// TIA Portal project "Synch Controller 20220313" (V15.1)

(* hardware
DEVICE "S71500/ET200MP station_1"  S7-1500 station
   slot 0: "导轨_0"  Rack  6ES7 590-1***0-0AA0
   slot 1: "PLC_1"  CPU 1516-3 PN/DP  6ES7 516-3AN01-0AB0  V2.6
      slot 3: "CPU 显示_1"  6ES7591-1BA00-0AA0
*)

// ===== PLC "PLC_1"  CPU 1516-3 PN/DP =====

VAR_GLOBAL   // PLC tag table "model"
   "left_cylinder_velocity" AT %MD200 : Real;
   "left_cylinder_position" AT %MD204 : Real;
   "right_cylinder_velocity" AT %MD208 : Real;
   "right_cylinder_position" AT %MD212 : Real;
   "left_cylinder_cmd[%]" AT %MD216 : Real;
   "right_cylinder_cmd[%]" AT %MD220 : Real;
   "model_run" AT %M100.0 : Bool;
   "left_cylinder_pos_init" AT %MD224 : Real;
   "right_cylinder_pos_init" AT %MD228 : Real;
END_VAR

VAR_GLOBAL   // PLC tag table "controller"
   "controller_run" AT %M300.1 : Bool;
   "ref_velocity" AT %MD400 : Real;
   "pos_loop_kp" AT %MD404 : Real;
   "pos_loop_Ti" AT %MD408 : Real;
   "vel_loop_kp" AT %MD412 : Real;
   "vel_loop_Ti" AT %MD416 : Real;
   "vel_loop_ff_kp" AT %MD420 : Real;
END_VAR

VAR_GLOBAL   // PLC tag table "test"
   "reset0" AT %M500.0 : Bool;
   "reset1" AT %M500.1 : Bool;
   "reset2" AT %M500.2 : Bool;
   "reset3" AT %M500.3 : Bool;
   "reset4" AT %M500.4 : Bool;
   "parameter1" AT %M500.6 : Bool;
   "parameter2" AT %M500.7 : Bool;
   "parameter3" AT %M501.0 : Bool;
   "parameter4" AT %M501.1 : Bool;
   "parameter5" AT %M501.2 : Bool;
   "autotest_run" AT %M500.5 : Bool;
   "seq_running" AT %M501.3 : Bool;
END_VAR

DATA_BLOCK "test_DB"   // DB3
{ S7_Optimized_Access := 'TRUE' }
VERSION : 0.1
// stored: InstanceOfName test
"test"
BEGIN
END_DATA_BLOCK

// folder: ctrl_synch/controller

DATA_BLOCK "controller_DB"   // DB9
{ S7_Optimized_Access := 'TRUE' }
VERSION : 0.1
// stored: InstanceOfName controller
"controller"
BEGIN
END_DATA_BLOCK

// folder: ctrl_synch/model

DATA_BLOCK "left_cylinder_DB"   // DB7
{ S7_Optimized_Access := 'TRUE' }
VERSION : 0.1
// stored: InstanceOfName cylinder
"cylinder"
BEGIN
END_DATA_BLOCK

DATA_BLOCK "right_cylinder_DB"   // DB8
{ S7_Optimized_Access := 'TRUE' }
VERSION : 0.1
// stored: InstanceOfName cylinder
"cylinder"
BEGIN
END_DATA_BLOCK

// folder: (top level)

FUNCTION_BLOCK "test"   // FB1, GRAPH_PLUS
{ S7_Optimized_Access := 'TRUE' }
VERSION : 0.1
   VAR_INPUT
      OFF_SQ : Bool := false;   // 关闭顺控器
      INIT_SQ : Bool := false;   // 将顺序设置为初始状态
      ACK_EF : Bool := false;   // 确认所有的错误和故障
      S_PREV : Bool := false;   // 在S_NO输出参数中显示前导步
      S_NEXT : Bool := false;   // 在S_NO输出参数中显示后续步。
      SW_AUTO : Bool := false;   // 自动模式
      SW_TAP : Bool := false;   // 半自动/转换条件切换
      SW_TOP : Bool := false;   // 半自动/忽略转换条件
      SW_MAN : Bool := false;   // 手动模式
      S_SEL : Int := 0;   // 选择要在 S_NO中输出的步。
      S_ON : Bool := false;   // 激活S_NO 中显示的步。
      S_OFF : Bool := false;   // 取消激活 S_NO 中标识的步
      T_PUSH : Bool := false;   // 允许在半自动模式下跳过转换条件。
   END_VAR
   VAR_OUTPUT
      S_NO : Int := 0;   // 步编号
      S_MORE : Bool := false;   // 更多步可用，并可在S_NO中显示。
      S_ACTIVE : Bool := false;   // 在S_NO 中显示的步是激活的。
      ERR_FLT : Bool := false;   // 互锁条件或监控条件组出错
      AUTO_ON : Bool := false;   // 当前为自动模式
      TAP_ON : Bool := false;   // 已启用SW_TAP模式。
      TOP_ON : Bool := false;   // 启用半自动模式/忽略转换条件。
      MAN_ON : Bool := false;   // 已启用手动模式。
      reset0 : Bool;   // initial status
      parameter1 : Bool;
      reset1 : Bool;
      parameter2 : Bool;
      reset2 : Bool;
      parameter3 : Bool;
      reset3 : Bool;
      parameter4 : Bool;
      reset4 : Bool;
      parameter5 : Bool;
   END_VAR
   VAR
      HMI_INFO : Array[0..8] of UInt;
      IF_PAR : G7_IfParPlus_V6;
      RT_DATA : G7_RTDataPlus_V6;   // 内部数据区
      Trans1 : G7_TransitionPlus_V6;   // 转换结构
      Trans2 : G7_TransitionPlus_V6;   // 转换结构
      Trans3 : G7_TransitionPlus_V6;   // 转换结构
      Trans4 : G7_TransitionPlus_V6;   // 转换结构
      Trans5 : G7_TransitionPlus_V6;   // 转换结构
      Trans6 : G7_TransitionPlus_V6;   // 转换结构
      Trans7 : G7_TransitionPlus_V6;   // 转换结构
      Trans8 : G7_TransitionPlus_V6;   // 转换结构
      Trans9 : G7_TransitionPlus_V6;   // 转换结构
      Trans10 : G7_TransitionPlus_V6;   // 转换结构
      Step1 : G7_StepPlus_V6;   // 步结构
      Step2 : G7_StepPlus_V6;   // 步结构
      Step3 : G7_StepPlus_V6;   // 步结构
      Step4 : G7_StepPlus_V6;   // 步结构
      Step5 : G7_StepPlus_V6;   // 步结构
      Step6 : G7_StepPlus_V6;   // 步结构
      Step7 : G7_StepPlus_V6;   // 步结构
      Step8 : G7_StepPlus_V6;   // 步结构
      Step9 : G7_StepPlus_V6;   // 步结构
      Step10 : G7_StepPlus_V6;   // 步结构
      SINI : Array[0..1] of USInt;
      LSTT : Array[0..9] of USInt;
      ATAJ : Array[0..9] of USInt;
      ATAB : Array[0..9] of USInt;
      PSTT : Array[0..9] of USInt;
      NSTT : Array[0..9] of USInt;
      ASSJ : Array[0..9] of USInt;
      ASSB : Array[0..9] of USInt;
      PTTS : Array[0..9] of USInt;
      NTTS : Array[0..9] of USInt;
      SW_SQTS : Array[0..9] of USInt;
      SWITCH : Array[0..0] of USInt;
      TVX : Array[0..1] of USInt;
      TTX : Array[0..1] of USInt;
      TSX : Array[0..1] of USInt;
      S00X : Array[0..1] of USInt;
      SOFFX : Array[0..1] of USInt;
      SONX : Array[0..1] of USInt;
      SAX : Array[0..1] of USInt;
      SERRX : Array[0..10] of USInt;
      SMX : Array[0..10] of USInt;
      S0X : Array[0..10] of USInt;
      S1X : Array[0..10] of USInt;
      IL_ALARM_INST : Diag_Alarm;
      SUP_ALARM_INST : Diag_Alarm;
      STEP_TIME_ALARM_INST : Diag_Alarm;
      IEC_TIMER_INST : IEC_TIMER;
      TRANSACTION_FLAG : Bool := false;
   END_VAR
   VAR CONSTANT
      MIN_INTERVAL : Time := T#10ms;
      MAX_INTERVAL : Time := T#40s;
      LAST_INTERVAL : Time := T#60s;
   END_VAR
   // SINI[0] := 2;
   // LSTT[0] := 255;
   // LSTT[1] := 255;
   // LSTT[2] := 255;
   // LSTT[3] := 255;
   // LSTT[4] := 255;
   // LSTT[5] := 255;
   // LSTT[6] := 255;
   // LSTT[7] := 255;
   // ATAJ[1] := 1;
   // ATAJ[2] := 2;
   // ATAJ[3] := 3;
   // ATAJ[4] := 4;
   // ATAJ[5] := 5;
   // ATAJ[6] := 6;
   // ATAJ[7] := 7;
   // ATAJ[8] := 8;
   // ATAB[1] := 1;
   // ATAB[2] := 2;
   // ATAB[3] := 3;
   // ATAB[4] := 4;
   // ATAB[5] := 5;
   // ATAB[6] := 6;
   // ATAB[7] := 7;
   // ATAB[8] := 8;
   // PSTT[1] := 1;
   // PSTT[2] := 2;
   // PSTT[3] := 3;
   // PSTT[4] := 4;
   // PSTT[5] := 5;
   // PSTT[6] := 6;
   // PSTT[7] := 7;
   // PSTT[8] := 8;
   // NSTT[0] := 1;
   // NSTT[1] := 2;
   // NSTT[2] := 3;
   // NSTT[3] := 4;
   // NSTT[4] := 5;
   // NSTT[5] := 6;
   // NSTT[6] := 7;
   // NSTT[7] := 8;
   // ASSJ[1] := 1;
   // ASSJ[2] := 2;
   // ASSJ[3] := 3;
   // ASSJ[4] := 4;
   // ASSJ[5] := 5;
   // ASSJ[6] := 6;
   // ASSJ[7] := 7;
   // ASSJ[8] := 8;
   // ASSB[1] := 1;
   // ASSB[2] := 2;
   // ASSB[3] := 3;
   // ASSB[4] := 4;
   // ASSB[5] := 5;
   // ASSB[6] := 6;
   // ASSB[7] := 7;
   // ASSB[8] := 8;
   // PTTS[0] := 255;
   // PTTS[2] := 1;
   // PTTS[3] := 2;
   // PTTS[4] := 3;
   // PTTS[5] := 4;
   // PTTS[6] := 5;
   // PTTS[7] := 6;
   // PTTS[8] := 7;
   // NTTS[1] := 1;
   // NTTS[2] := 2;
   // NTTS[3] := 3;
   // NTTS[4] := 4;
   // NTTS[5] := 5;
   // NTTS[6] := 6;
   // NTTS[7] := 7;
   // NTTS[8] := 8;
   // TVX[0] := 16#1;
   // TTX[0] := 16#1;
   // TSX[0] := 16#1;
   // S00X[0] := 16#1;
   // SOFFX[0] := 16#1;
   // SONX[0] := 16#1;
   // SAX[0] := 16#1;
   // SERRX[0] := 16#1;
   // SMX[0] := 16#1;
   // S0X[0] := 16#1;
   // S1X[0] := 16#1;
   // LSTT[8] := 255;
   // ATAJ[9] := 9;
   // ATAB[9] := 9;
   // PSTT[9] := 9;
   // NSTT[8] := 9;
   // ASSJ[9] := 9;
   // ASSB[9] := 9;
   // PTTS[9] := 8;
   // NTTS[9] := 9;
BEGIN
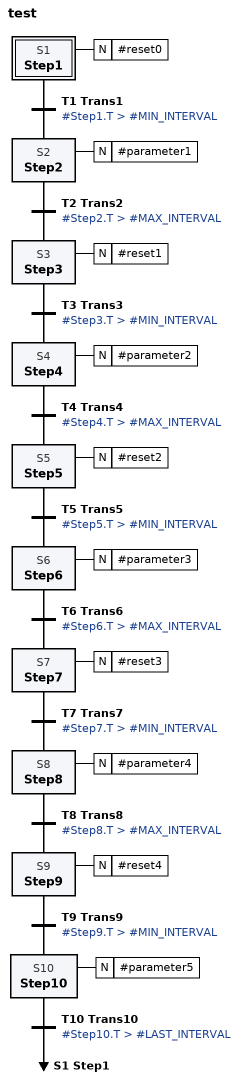
   // sequencer 1
   INITIAL_STEP Step1:   // S1, max time T#10S, warning time T#7S
              N    #reset0
   END_STEP
   TRANSITION Trans1 FROM Step1 TO Step2   // T1
      := #Step1.T > #MIN_INTERVAL;
   END_TRANSITION
   STEP Step2:   // S2, max time T#10S, warning time T#7S
              N    #parameter1
   END_STEP
   TRANSITION Trans2 FROM Step2 TO Step3   // T2
      := #Step2.T > #MAX_INTERVAL;
   END_TRANSITION
   STEP Step3:   // S3, max time T#10S, warning time T#7S
              N    #reset1
   END_STEP
   TRANSITION Trans3 FROM Step3 TO Step4   // T3
      := #Step3.T > #MIN_INTERVAL;
   END_TRANSITION
   STEP Step4:   // S4, max time T#10S, warning time T#7S
              N    #parameter2
   END_STEP
   TRANSITION Trans4 FROM Step4 TO Step5   // T4
      := #Step4.T > #MAX_INTERVAL;
   END_TRANSITION
   STEP Step5:   // S5, max time T#10S, warning time T#7S
              N    #reset2
   END_STEP
   TRANSITION Trans5 FROM Step5 TO Step6   // T5
      := #Step5.T > #MIN_INTERVAL;
   END_TRANSITION
   STEP Step6:   // S6, max time T#10S, warning time T#7S
              N    #parameter3
   END_STEP
   TRANSITION Trans6 FROM Step6 TO Step7   // T6
      := #Step6.T > #MAX_INTERVAL;
   END_TRANSITION
   STEP Step7:   // S7, max time T#10S, warning time T#7S
              N    #reset3
   END_STEP
   TRANSITION Trans7 FROM Step7 TO Step8   // T7
      := #Step7.T > #MIN_INTERVAL;
   END_TRANSITION
   STEP Step8:   // S8, max time T#10S, warning time T#7S
              N    #parameter4
   END_STEP
   TRANSITION Trans8 FROM Step8 TO Step9   // T8
      := #Step8.T > #MAX_INTERVAL;
   END_TRANSITION
   STEP Step9:   // S9, max time T#10S, warning time T#7S
              N    #reset4
   END_STEP
   TRANSITION Trans9 FROM Step9 TO Step10   // T9
      := #Step9.T > #MIN_INTERVAL;
   END_TRANSITION
   STEP Step10:   // S10, max time T#10S, warning time T#7S
              N    #parameter5
   END_STEP
   TRANSITION Trans10 FROM Step10 TO Step1   // T10, jump
      := #Step10.T > #LAST_INTERVAL;
   END_TRANSITION
END_FUNCTION_BLOCK

ORGANIZATION_BLOCK "Main"   // OB1, LAD, ProgramCycle
TITLE = "Main Program Sweep (Cycle)"
{ S7_Optimized_Access := 'TRUE' }
VERSION : 0.1
   VAR_INPUT
      Initial_Call : Bool;   // Initial call of this OB
      Remanence : Bool;   // =True, if remanent data are available
   END_VAR
BEGIN

REGION Network 1
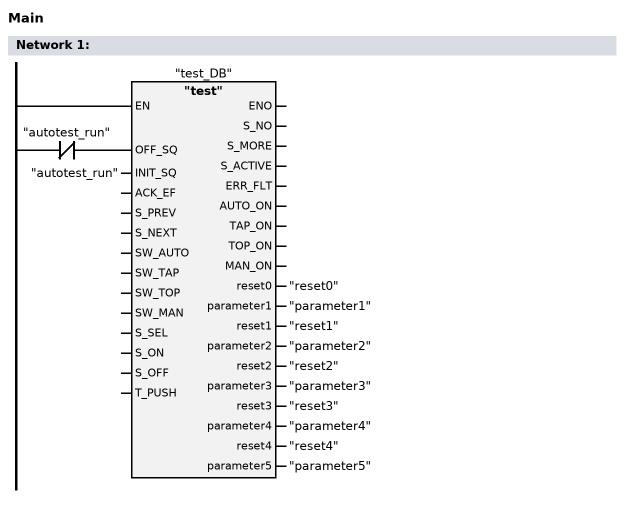
   RUNG wire#powerrail
      "test_DB"(OFF_SQ := wire#w1, INIT_SQ := "autotest_run", ACK_EF :=, S_PREV :=, S_NEXT :=, SW_AUTO :=, SW_TAP :=, SW_TOP :=, SW_MAN :=, S_SEL :=, S_ON :=, S_OFF :=, T_PUSH :=, S_NO =>, S_MORE =>, S_ACTIVE =>, ERR_FLT =>, AUTO_ON =>, TAP_ON =>, TOP_ON =>, MAN_ON =>, reset0 => "reset0", parameter1 => "parameter1", reset1 => "reset1", parameter2 => "parameter2", reset2 => "reset2", parameter3 => "parameter3", reset3 => "reset3", parameter4 => "parameter4", reset4 => "reset4", parameter5 => "parameter5")
   END_RUNG
   RUNG wire#powerrail
      I_Contact( "autotest_run" )
   END_RUNG wire#w1
   // the same network as SCL:
   "test_DB"(OFF_SQ := NOT "autotest_run",   // "test"
             INIT_SQ := "autotest_run",
             reset0 => "reset0",
             parameter1 => "parameter1",
             reset1 => "reset1",
             parameter2 => "parameter2",
             reset2 => "reset2",
             parameter3 => "parameter3",
             reset3 => "reset3",
             parameter4 => "parameter4",
             reset4 => "reset4",
             parameter5 => "parameter5");
END_REGION

REGION Network 2 (SCL): test-1
   // rated speed of cylinder = 50mm/s [100% openning of valve]
   // only position loop
   // IF ("reset0" OR
   //     "reset1" OR
   //     "reset2" OR
   //     "reset3" OR
   //     "reset4")OR
   //     NOT "autotest_run"
   // THEN
   //     "left_cylinder_pos_init" :=1100.0;
   //     "right_cylinder_pos_init" :=900.0;
   //     "ref_velocity" := 0.0;
   //     "model_run" := FALSE;
   //     "controller_run" := FALSE;
   // END_IF;

   // IF "parameter1" THEN
   //     "model_run" := TRUE;
   //     "controller_run" := TRUE;

   //     "ref_velocity" := 0.0;
   //     "pos_loop_kp" := 1.0;
   //     "pos_loop_Ti" := 0.0;
   //     "vel_loop_kp" := 0.0;
   //     "vel_loop_Ti" := 0.0;
   //     "vel_loop_ff_kp" := 1.0;

   // END_IF;


   // IF "parameter2" THEN
   //     "model_run" := TRUE;
   //     "controller_run" := TRUE;

   //     "ref_velocity" := 0.0;
   //     "pos_loop_kp" := 5.0;
   //     "pos_loop_Ti" := 0.0;
   //     "vel_loop_kp" := 0.0;
   //     "vel_loop_Ti" := 0.0;
   //     "vel_loop_ff_kp" := 1.0;

   // END_IF;

   // IF "parameter3" THEN
   //     "model_run" := TRUE;
   //     "controller_run" := TRUE;

   //     "ref_velocity" := 0.0;
   //     "pos_loop_kp" := 10.0;
   //     "pos_loop_Ti" := 0.0;
   //     "vel_loop_kp" := 0.0;
   //     "vel_loop_Ti" := 0.0;
   //     "vel_loop_ff_kp" := 1.0;

   // END_IF;

   // IF "parameter4" THEN
   //     "model_run" := TRUE;
   //     "controller_run" := TRUE;

   //     "ref_velocity" := 0.0;
   //     "pos_loop_kp" := 15.0;
   //     "pos_loop_Ti" := 0.0;
   //     "vel_loop_kp" := 0.0;
   //     "vel_loop_Ti" := 0.0;
   //     "vel_loop_ff_kp" := 1.0;

   // END_IF;

   // IF "parameter5" THEN
   //     "model_run" := TRUE;
   //     "controller_run" := TRUE;

   //     "ref_velocity" := 0.0;
   //     "pos_loop_kp" := 20.0;
   //     "pos_loop_Ti" := 0.0;
   //     "vel_loop_kp" := 0.0;
   //     "vel_loop_Ti" := 0.0;
   //     "vel_loop_ff_kp" := 1.0;

   // END_IF;
END_REGION

REGION Network 3 (SCL): test-2
   // rated speed of cylinder = 50mm/s [100% openning of valve]
   // position loop+velocity loop
   // IF ("reset0" OR
   //     "reset1" OR
   //     "reset2" OR
   //     "reset3" OR
   //     "reset4")OR
   //     NOT "autotest_run"
   // THEN
   //     "left_cylinder_pos_init" :=1100.0;
   //     "right_cylinder_pos_init" :=900.0;
   //     "ref_velocity" := 0.0;
   //     "model_run" := FALSE;
   //     "controller_run" := FALSE;
   // END_IF;
   // // 
   // IF "parameter1" THEN
   //     "model_run" := TRUE;
   //     "controller_run" := TRUE;

   //     "ref_velocity" := 0.0;
   //     "pos_loop_kp" := 1.0;
   //     "pos_loop_Ti" := 0.0;
   //     "vel_loop_kp" := 1.0;
   //     "vel_loop_Ti" := 0.0;
   //     "vel_loop_ff_kp" := 0.0;

   // END_IF;

   // // 
   // IF "parameter2" THEN
   //     "model_run" := TRUE;
   //     "controller_run" := TRUE;

   //     "ref_velocity" := 0.0;
   //     "pos_loop_kp" := 5.0;
   //     "pos_loop_Ti" := 0.0;
   //     "vel_loop_kp" := 1.0;
   //     "vel_loop_Ti" := 0.0;
   //     "vel_loop_ff_kp" := 0.0;

   // END_IF;
   // // 
   // IF "parameter3" THEN
   //     "model_run" := TRUE;
   //     "controller_run" := TRUE;

   //     "ref_velocity" := 0.0;
   //     "pos_loop_kp" := 10.0;
   //     "pos_loop_Ti" := 0.0;
   //     "vel_loop_kp" := 1.0;
   //     "vel_loop_Ti" := 0.0;
   //     "vel_loop_ff_kp" := 0.0;

   // END_IF;
   // //
   // IF "parameter4" THEN
   //     "model_run" := TRUE;
   //     "controller_run" := TRUE;

   //     "ref_velocity" := 0.0;
   //     "pos_loop_kp" := 15.0;
   //     "pos_loop_Ti" := 0.0;
   //     "vel_loop_kp" := 1.0;
   //     "vel_loop_Ti" := 0.0;
   //     "vel_loop_ff_kp" := 0.0;

   // END_IF;
   // //
   // IF "parameter5" THEN
   //     "model_run" := TRUE;
   //     "controller_run" := TRUE;

   //     "ref_velocity" := 0.0;
   //     "pos_loop_kp" := 20.0;
   //     "pos_loop_Ti" := 0.0;
   //     "vel_loop_kp" := 1.0;
   //     "vel_loop_Ti" := 0.0;
   //     "vel_loop_ff_kp" := 0.0;

   // END_IF;
END_REGION

REGION Network 4 (SCL): test-3
   // rated speed of cylinder = 50mm/s [100% openning of valve]
   // position loop+velocity loop+FF
   // IF ("reset0" OR
   //     "reset1" OR
   //     "reset2" OR
   //     "reset3" OR
   //     "reset4")OR
   //     NOT "autotest_run"
   // THEN
   //     "left_cylinder_pos_init" :=1100.0;
   //     "right_cylinder_pos_init" :=900.0;
   //     "ref_velocity" := 0.0;
   //     "model_run" := FALSE;
   //     "controller_run" := FALSE;
   // END_IF;
   // // 
   // IF "parameter1" THEN
   //     "model_run" := TRUE;
   //     "controller_run" := TRUE;

   //     "ref_velocity" := 0.0;
   //     "pos_loop_kp" := 1.0;
   //     "pos_loop_Ti" := 0.0;
   //     "vel_loop_kp" := 1.0;
   //     "vel_loop_Ti" := 0.0;
   //     "vel_loop_ff_kp" := 1.0;

   // END_IF;

   // // 
   // IF "parameter2" THEN
   //     "model_run" := TRUE;
   //     "controller_run" := TRUE;

   //     "ref_velocity" := 0.0;
   //     "pos_loop_kp" := 5.0;
   //     "pos_loop_Ti" := 0.0;
   //     "vel_loop_kp" := 1.0;
   //     "vel_loop_Ti" := 0.0;
   //     "vel_loop_ff_kp" := 1.0;

   // END_IF;
   // // 
   // IF "parameter3" THEN
   //     "model_run" := TRUE;
   //     "controller_run" := TRUE;

   //     "ref_velocity" := 0.0;
   //     "pos_loop_kp" := 10.0;
   //     "pos_loop_Ti" := 0.0;
   //     "vel_loop_kp" := 1.0;
   //     "vel_loop_Ti" := 0.0;
   //     "vel_loop_ff_kp" := 1.0;

   // END_IF;
   // //
   // IF "parameter4" THEN
   //     "model_run" := TRUE;
   //     "controller_run" := TRUE;

   //     "ref_velocity" := 0.0;
   //     "pos_loop_kp" := 15.0;
   //     "pos_loop_Ti" := 0.0;
   //     "vel_loop_kp" := 1.0;
   //     "vel_loop_Ti" := 0.0;
   //     "vel_loop_ff_kp" := 1.0;

   // END_IF;
   // //
   // IF "parameter5" THEN
   //     "model_run" := TRUE;
   //     "controller_run" := TRUE;

   //     "ref_velocity" := 0.0;
   //     "pos_loop_kp" := 20.0;
   //     "pos_loop_Ti" := 0.0;
   //     "vel_loop_kp" := 1.0;
   //     "vel_loop_Ti" := 0.0;
   //     "vel_loop_ff_kp" := 1.0;

   // END_IF;
END_REGION

REGION Network 5 (SCL): test-4
   // velocity loop
   // IF ("reset0" OR
   //     "reset1" OR
   //     "reset2" OR
   //     "reset3" OR
   //     "reset4")OR
   //     NOT "autotest_run"
   // THEN
   //     "left_cylinder_pos_init" :=1000.0;
   //     "right_cylinder_pos_init" :=1000.0;
   //     "ref_velocity" := 0.0;
   //     "model_run" := FALSE;
   //     "controller_run" := FALSE;
   // END_IF;
   // // 
   // IF "parameter1" THEN
   //     "model_run" := TRUE;
   //     "controller_run" := TRUE;

   //     "ref_velocity" := 40.0;
   //     "pos_loop_kp" := 10.0;
   //     "pos_loop_Ti" := 0.0;
   //     "vel_loop_kp" := 1.0;
   //     "vel_loop_Ti" := 0.0;
   //     "vel_loop_ff_kp" := 0.0;

   // END_IF;

   // // 
   // IF "parameter2" THEN
   //     "model_run" := TRUE;
   //     "controller_run" := TRUE;

   //     "ref_velocity" := 40.0;
   //     "pos_loop_kp" := 10.0;
   //     "pos_loop_Ti" := 0.0;
   //     "vel_loop_kp" := 2.0;
   //     "vel_loop_Ti" := 0.0;
   //     "vel_loop_ff_kp" := 1.0;

   // END_IF;
   // // 
   // IF "parameter3" THEN
   //     "model_run" := TRUE;
   //     "controller_run" := TRUE;

   //     "ref_velocity" := 40.0;
   //     "pos_loop_kp" := 10.0;
   //     "pos_loop_Ti" := 0.0;
   //     "vel_loop_kp" := 5.0;
   //     "vel_loop_Ti" := 0.0;
   //     "vel_loop_ff_kp" := 0.0;

   // END_IF;
   // //
   // IF "parameter4" THEN
   //     "model_run" := TRUE;
   //     "controller_run" := TRUE;

   //     "ref_velocity" := 40.0;
   //     "pos_loop_kp" := 10.0;
   //     "pos_loop_Ti" := 0.0;
   //     "vel_loop_kp" := 10.0;
   //     "vel_loop_Ti" := 0.0;
   //     "vel_loop_ff_kp" := 0.0;

   // END_IF;
   // //
   // IF "parameter5" THEN
   //     "model_run" := TRUE;
   //     "controller_run" := TRUE;

   //     "ref_velocity" := 40.0;
   //     "pos_loop_kp" := 10.0;
   //     "pos_loop_Ti" := 0.0;
   //     "vel_loop_kp" := 20.0;
   //     "vel_loop_Ti" := 0.0;
   //     "vel_loop_ff_kp" := 0.0;

   // END_IF;
END_REGION

REGION Network 6 (SCL): test-5
   // velocity loop
   // IF ("reset0" OR
   //     "reset1" OR
   //     "reset2" OR
   //     "reset3" OR
   //     "reset4")OR
   //     NOT "autotest_run"
   // THEN
   //     "left_cylinder_pos_init" :=1000.0;
   //     "right_cylinder_pos_init" :=1000.0;
   //     "ref_velocity" := 0.0;
   //     "model_run" := FALSE;
   //     "controller_run" := FALSE;
   // END_IF;
   // // 
   // IF "parameter1" THEN
   //     "model_run" := TRUE;
   //     "controller_run" := TRUE;

   //     "ref_velocity" := 40.0;
   //     "pos_loop_kp" := 10.0;
   //     "pos_loop_Ti" := 0.0;
   //     "vel_loop_kp" := 1.0;
   //     "vel_loop_Ti" := 1.0;
   //     "vel_loop_ff_kp" := 0.0;

   // END_IF;

   // // 
   // IF "parameter2" THEN
   //     "model_run" := TRUE;
   //     "controller_run" := TRUE;

   //     "ref_velocity" := 40.0;
   //     "pos_loop_kp" := 10.0;
   //     "pos_loop_Ti" := 0.0;
   //     "vel_loop_kp" := 2.0;
   //     "vel_loop_Ti" := 1.0;
   //     "vel_loop_ff_kp" := 1.0;

   // END_IF;
   // // 
   // IF "parameter3" THEN
   //     "model_run" := TRUE;
   //     "controller_run" := TRUE;

   //     "ref_velocity" := 40.0;
   //     "pos_loop_kp" := 10.0;
   //     "pos_loop_Ti" := 0.0;
   //     "vel_loop_kp" := 5.0;
   //     "vel_loop_Ti" := 1.0;
   //     "vel_loop_ff_kp" := 0.0;

   // END_IF;
   // //
   // IF "parameter4" THEN
   //     "model_run" := TRUE;
   //     "controller_run" := TRUE;

   //     "ref_velocity" := 40.0;
   //     "pos_loop_kp" := 10.0;
   //     "pos_loop_Ti" := 0.0;
   //     "vel_loop_kp" := 10.0;
   //     "vel_loop_Ti" := 1.0;
   //     "vel_loop_ff_kp" := 0.0;

   // END_IF;
   // //
   // IF "parameter5" THEN
   //     "model_run" := TRUE;
   //     "controller_run" := TRUE;

   //     "ref_velocity" := 40.0;
   //     "pos_loop_kp" := 10.0;
   //     "pos_loop_Ti" := 0.0;
   //     "vel_loop_kp" := 20.0;
   //     "vel_loop_Ti" := 1.0;
   //     "vel_loop_ff_kp" := 0.0;

   // END_IF;
END_REGION

REGION Network 7 (SCL): test-5
   // velocity loop
   // IF ("reset0" OR
   //     "reset1" OR
   //     "reset2" OR
   //     "reset3" OR
   //     "reset4")OR
   //     NOT "autotest_run"
   // THEN
   //     "left_cylinder_pos_init" :=1000.0;
   //     "right_cylinder_pos_init" :=1000.0;
   //     "ref_velocity" := 0.0;
   //     "model_run" := FALSE;
   //     "controller_run" := FALSE;
   // END_IF;

   // IF "parameter1" THEN
   //     "model_run" := TRUE;
   //     "controller_run" := TRUE;

   //     "ref_velocity" := 40.0;
   //     "pos_loop_kp" := 10.0;
   //     "pos_loop_Ti" := 0.0;
   //     "vel_loop_kp" := 1.0;
   //     "vel_loop_Ti" := 10.0;
   //     "vel_loop_ff_kp" := 0.0;

   // END_IF;


   // IF "parameter2" THEN
   //     "model_run" := TRUE;
   //     "controller_run" := TRUE;

   //     "ref_velocity" := 40.0;
   //     "pos_loop_kp" := 10.0;
   //     "pos_loop_Ti" := 0.0;
   //     "vel_loop_kp" := 2.0;
   //     "vel_loop_Ti" := 10.0;
   //     "vel_loop_ff_kp" := 0.0;

   // END_IF;

   // IF "parameter3" THEN
   //     "model_run" := TRUE;
   //     "controller_run" := TRUE;

   //     "ref_velocity" := 40.0;
   //     "pos_loop_kp" := 10.0;
   //     "pos_loop_Ti" := 0.0;
   //     "vel_loop_kp" := 5.0;
   //     "vel_loop_Ti" := 10.0;
   //     "vel_loop_ff_kp" := 0.0;

   // END_IF;

   // IF "parameter4" THEN
   //     "model_run" := TRUE;
   //     "controller_run" := TRUE;

   //     "ref_velocity" := 40.0;
   //     "pos_loop_kp" := 10.0;
   //     "pos_loop_Ti" := 0.0;
   //     "vel_loop_kp" := 10.0;
   //     "vel_loop_Ti" := 10.0;
   //     "vel_loop_ff_kp" := 0.0;

   // END_IF;

   // IF "parameter5" THEN
   //     "model_run" := TRUE;
   //     "controller_run" := TRUE;

   //     "ref_velocity" := 40.0;
   //     "pos_loop_kp" := 10.0;
   //     "pos_loop_Ti" := 0.0;
   //     "vel_loop_kp" := 20.0;
   //     "vel_loop_Ti" := 10.0;
   //     "vel_loop_ff_kp" := 0.0;

   // END_IF;
END_REGION

REGION Network 8 (SCL): test-7
   // velocity loop
   // IF ("reset0" OR
   //     "reset1" OR
   //     "reset2" OR
   //     "reset3" OR
   //     "reset4")OR
   //     NOT "autotest_run"
   // THEN
   //     "left_cylinder_pos_init" :=1000.0;
   //     "right_cylinder_pos_init" :=1000.0;
   //     "ref_velocity" := 0.0;
   //     "model_run" := FALSE;
   //     "controller_run" := FALSE;
   // END_IF;
   // // 
   // IF "parameter1" THEN
   //     "model_run" := TRUE;
   //     "controller_run" := TRUE;

   //     "ref_velocity" := 40.0;
   //     "pos_loop_kp" := 10.0;
   //     "pos_loop_Ti" := 0.0;
   //     "vel_loop_kp" := 1.0;
   //     "vel_loop_Ti" := 1.0;
   //     "vel_loop_ff_kp" := 0.0;

   // END_IF;

   // // 
   // IF "parameter2" THEN
   //     "model_run" := TRUE;
   //     "controller_run" := TRUE;

   //     "ref_velocity" := 40.0;
   //     "pos_loop_kp" := 10.0;
   //     "pos_loop_Ti" := 0.0;
   //     "vel_loop_kp" := 2.0;
   //     "vel_loop_Ti" := 1.0;
   //     "vel_loop_ff_kp" := 0.0;

   // END_IF;
   // // 
   // IF "parameter3" THEN
   //     "model_run" := TRUE;
   //     "controller_run" := TRUE;

   //     "ref_velocity" := 40.0;
   //     "pos_loop_kp" := 10.0;
   //     "pos_loop_Ti" := 0.0;
   //     "vel_loop_kp" := 2.0;
   //     "vel_loop_Ti" := 2.0;
   //     "vel_loop_ff_kp" := 0.0;

   // END_IF;
   // //
   // IF "parameter4" THEN
   //     "model_run" := TRUE;
   //     "controller_run" := TRUE;

   //     "ref_velocity" := 40.0;
   //     "pos_loop_kp" := 10.0;
   //     "pos_loop_Ti" := 0.0;
   //     "vel_loop_kp" := 5.0;
   //     "vel_loop_Ti" := 5.0;
   //     "vel_loop_ff_kp" := 0.0;

   // END_IF;
   // //
   // IF "parameter5" THEN
   //     "model_run" := TRUE;
   //     "controller_run" := TRUE;

   //     "ref_velocity" := 40.0;
   //     "pos_loop_kp" := 10.0;
   //     "pos_loop_Ti" := 0.0;
   //     "vel_loop_kp" := 5.0;
   //     "vel_loop_Ti" := 10.0;
   //     "vel_loop_ff_kp" := 0.0;

   // END_IF;
END_REGION

REGION Network 9 (SCL): test-9
   // velocity loop
   // IF ("reset0" OR
   //     "reset1" OR
   //     "reset2" OR
   //     "reset3" OR
   //     "reset4")OR
   //     NOT "autotest_run"
   // THEN
   //     "left_cylinder_pos_init" :=1100.0;
   //     "right_cylinder_pos_init" :=900.0;
   //     "ref_velocity" := 0.0;
   //     "model_run" := FALSE;
   //     "controller_run" := FALSE;
   // END_IF;
   // // 
   // IF "parameter1" THEN
   //     "model_run" := TRUE;
   //     "controller_run" := TRUE;

   //     "ref_velocity" := 0.0;
   //     "pos_loop_kp" := 10.0;
   //     "pos_loop_Ti" := 0.0;
   //     "vel_loop_kp" := 1.0;
   //     "vel_loop_Ti" := 1.0;
   //     "vel_loop_ff_kp" := 0.0;

   // END_IF;

   // // 
   // IF "parameter2" THEN
   //     "model_run" := TRUE;
   //     "controller_run" := TRUE;

   //     "ref_velocity" := 0.0;
   //     "pos_loop_kp" := 10.0;
   //     "pos_loop_Ti" := 0.0;
   //     "vel_loop_kp" := 2.0;
   //     "vel_loop_Ti" := 1.0;
   //     "vel_loop_ff_kp" := 0.0;

   // END_IF;
   // // 
   // IF "parameter3" THEN
   //     "model_run" := TRUE;
   //     "controller_run" := TRUE;

   //     "ref_velocity" := 0.0;
   //     "pos_loop_kp" := 10.0;
   //     "pos_loop_Ti" := 0.0;
   //     "vel_loop_kp" := 2.0;
   //     "vel_loop_Ti" := 2.0;
   //     "vel_loop_ff_kp" := 0.0;

   // END_IF;
   // //
   // IF "parameter4" THEN
   //     "model_run" := TRUE;
   //     "controller_run" := TRUE;

   //     "ref_velocity" := 0.0;
   //     "pos_loop_kp" := 10.0;
   //     "pos_loop_Ti" := 0.0;
   //     "vel_loop_kp" := 5.0;
   //     "vel_loop_Ti" := 5.0;
   //     "vel_loop_ff_kp" := 0.0;

   // END_IF;
   // //
   // IF "parameter5" THEN
   //     "model_run" := TRUE;
   //     "controller_run" := TRUE;

   //     "ref_velocity" := 0.0;
   //     "pos_loop_kp" := 10.0;
   //     "pos_loop_Ti" := 0.0;
   //     "vel_loop_kp" := 5.0;
   //     "vel_loop_Ti" := 10.0;
   //     "vel_loop_ff_kp" := 0.0;

   // END_IF;
END_REGION

REGION Network 10 (SCL): test-10
   // velocity loop
   // IF ("reset0" OR
   //     "reset1" OR
   //     "reset2" OR
   //     "reset3" OR
   //     "reset4")OR
   //     NOT "autotest_run"
   // THEN
   //     "left_cylinder_pos_init" :=1100.0;
   //     "right_cylinder_pos_init" :=900.0;
   //     "ref_velocity" := 0.0;
   //     "model_run" := FALSE;
   //     "controller_run" := FALSE;
   // END_IF;
   // // 
   // IF "parameter1" THEN
   //     "model_run" := TRUE;
   //     "controller_run" := TRUE;

   //     "ref_velocity" := 0.0;
   //     "pos_loop_kp" := 5.0;
   //     "pos_loop_Ti" := 0.0;
   //     "vel_loop_kp" := 2.0;
   //     "vel_loop_Ti" := 5.0;
   //     "vel_loop_ff_kp" := 0.0;

   // END_IF;

   // // 
   // IF "parameter2" THEN
   //     "model_run" := TRUE;
   //     "controller_run" := TRUE;

   //     "ref_velocity" := 0.0;
   //     "pos_loop_kp" := 5.0;
   //     "pos_loop_Ti" := 0.0;
   //     "vel_loop_kp" := 2.0;
   //     "vel_loop_Ti" := 10.0;
   //     "vel_loop_ff_kp" := 0.0;

   // END_IF;
   // // 
   // IF "parameter3" THEN
   //     "model_run" := TRUE;
   //     "controller_run" := TRUE;

   //     "ref_velocity" := 0.0;
   //     "pos_loop_kp" := 2.0;
   //     "pos_loop_Ti" := 0.0;
   //     "vel_loop_kp" := 2.0;
   //     "vel_loop_Ti" := 5.0;
   //     "vel_loop_ff_kp" := 0.0;

   // END_IF;
   // //
   // IF "parameter4" THEN
   //     "model_run" := TRUE;
   //     "controller_run" := TRUE;

   //     "ref_velocity" := 0.0;
   //     "pos_loop_kp" := 2.0;
   //     "pos_loop_Ti" := 0.0;
   //     "vel_loop_kp" := 2.0;
   //     "vel_loop_Ti" := 10.0;
   //     "vel_loop_ff_kp" := 0.0;

   // END_IF;
   // //
   // IF "parameter5" THEN
   //     "model_run" := TRUE;
   //     "controller_run" := TRUE;

   //     "ref_velocity" := 0.0;
   //     "pos_loop_kp" := 2.0;
   //     "pos_loop_Ti" := 0.0;
   //     "vel_loop_kp" := 2.0;
   //     "vel_loop_Ti" := 10.0;
   //     "vel_loop_ff_kp" := 0.0;

   // END_IF;
END_REGION

REGION Network 11 (SCL): test-11
   // velocity loop
   // IF ("reset0" OR
   //     "reset1" OR
   //     "reset2" OR
   //     "reset3" OR
   //     "reset4")OR
   //     NOT "autotest_run"
   // THEN
   //     "left_cylinder_pos_init" :=1100.0;
   //     "right_cylinder_pos_init" :=900.0;
   //     "ref_velocity" := 0.0;
   //     "model_run" := FALSE;
   //     "controller_run" := FALSE;
   // END_IF;
   // // 
   // IF "parameter1" THEN
   //     "model_run" := TRUE;
   //     "controller_run" := TRUE;

   //     "ref_velocity" := 0.0;
   //     "pos_loop_kp" := 1.0;
   //     "pos_loop_Ti" := 0.0;
   //     "vel_loop_kp" := 1.0;
   //     "vel_loop_Ti" := 10.0;
   //     "vel_loop_ff_kp" := 1.0;

   // END_IF;

   // // 
   // IF "parameter2" THEN
   //     "model_run" := TRUE;
   //     "controller_run" := TRUE;

   //     "ref_velocity" := 0.0;
   //     "pos_loop_kp" := 1.0;
   //     "pos_loop_Ti" := 0.0;
   //     "vel_loop_kp" := 1.0;
   //     "vel_loop_Ti" := 10.0;
   //     "vel_loop_ff_kp" := 2.0;

   // END_IF;
   // // 
   // IF "parameter3" THEN
   //     "model_run" := TRUE;
   //     "controller_run" := TRUE;

   //     "ref_velocity" := 0.0;
   //     "pos_loop_kp" := 1.0;
   //     "pos_loop_Ti" := 0.0;
   //     "vel_loop_kp" := 1.0;
   //     "vel_loop_Ti" := 10.0;
   //     "vel_loop_ff_kp" := 5.0;

   // END_IF;
   // //
   // IF "parameter4" THEN
   //     "model_run" := TRUE;
   //     "controller_run" := TRUE;

   //     "ref_velocity" := 0.0;
   //     "pos_loop_kp" := 1.0;
   //     "pos_loop_Ti" := 0.0;
   //     "vel_loop_kp" := 1.0;
   //     "vel_loop_Ti" := 10.0;
   //     "vel_loop_ff_kp" := 10.0;

   // END_IF;
   // //
   // IF "parameter5" THEN
   //     "model_run" := TRUE;
   //     "controller_run" := TRUE;

   //     "ref_velocity" := 0.0;
   //     "pos_loop_kp" := 1.0;
   //     "pos_loop_Ti" := 10.0;
   //     "vel_loop_kp" := 1.0;
   //     "vel_loop_Ti" := 10.0;
   //     "vel_loop_ff_kp" := 0.0;

   // END_IF;
END_REGION

REGION Network 12 (SCL): test-12
   // velocity loop
   // IF ("reset0" OR
   //     "reset1" OR
   //     "reset2" OR
   //     "reset3" OR
   //     "reset4")OR
   //     NOT "autotest_run"
   // THEN
   //     "left_cylinder_pos_init" :=1100.0;
   //     "right_cylinder_pos_init" :=900.0;
   //     "ref_velocity" := 0.0;
   //     "model_run" := FALSE;
   //     "controller_run" := FALSE;
   // END_IF;
   // // 
   // IF "parameter1" THEN
   //     "model_run" := TRUE;
   //     "controller_run" := TRUE;

   //     "ref_velocity" := 0.0;
   //     "pos_loop_kp" := 0.5;
   //     "pos_loop_Ti" := 10.0;
   //     "vel_loop_kp" := 1.0;
   //     "vel_loop_Ti" := 10.0;
   //     "vel_loop_ff_kp" := 10.0;

   // END_IF;

   // // 
   // IF "parameter2" THEN
   //     "model_run" := TRUE;
   //     "controller_run" := TRUE;

   //     "ref_velocity" := 0.0;
   //     "pos_loop_kp" := 0.5;
   //     "pos_loop_Ti" := 20.0;
   //     "vel_loop_kp" := 1.0;
   //     "vel_loop_Ti" := 10.0;
   //     "vel_loop_ff_kp" := 10.0;

   // END_IF;
   // // 
   // IF "parameter3" THEN
   //     "model_run" := TRUE;
   //     "controller_run" := TRUE;

   //     "ref_velocity" := 0.0;
   //     "pos_loop_kp" := 0.5;
   //     "pos_loop_Ti" := 30.0;
   //     "vel_loop_kp" := 1.0;
   //     "vel_loop_Ti" := 10.0;
   //     "vel_loop_ff_kp" := 10.0;

   // END_IF;
   // //
   // IF "parameter4" THEN
   //     "model_run" := TRUE;
   //     "controller_run" := TRUE;

   //     "ref_velocity" := 0.0;
   //     "pos_loop_kp" := 0.5;
   //     "pos_loop_Ti" := 40.0;
   //     "vel_loop_kp" := 1.0;
   //     "vel_loop_Ti" := 10.0;
   //     "vel_loop_ff_kp" := 10.0;

   // END_IF;
   // //
   // IF "parameter5" THEN
   //     "model_run" := TRUE;
   //     "controller_run" := TRUE;

   //     "ref_velocity" := 0.0;
   //     "pos_loop_kp" := 0.5;
   //     "pos_loop_Ti" := 50.0;
   //     "vel_loop_kp" := 1.0;
   //     "vel_loop_Ti" := 10.0;
   //     "vel_loop_ff_kp" := 10.0;

   // END_IF;
END_REGION

REGION Network 13 (SCL): test-13
   // velocity loop
   // IF ("reset0" OR
   //     "reset1" OR
   //     "reset2" OR
   //     "reset3" OR
   //     "reset4")OR
   //     NOT "autotest_run"
   // THEN
   //     "left_cylinder_pos_init" :=1100.0;
   //     "right_cylinder_pos_init" :=900.0;
   //     "ref_velocity" := 0.0;
   //     "model_run" := FALSE;
   //     "controller_run" := FALSE;
   // END_IF;
   // // 
   // IF "parameter1" THEN
   //     "model_run" := TRUE;
   //     "controller_run" := TRUE;

   //     "ref_velocity" := 0.0;
   //     "pos_loop_kp" := 0.5;
   //     "pos_loop_Ti" := 0.0;
   //     "vel_loop_kp" := 1.0;
   //     "vel_loop_Ti" := 10.0;
   //     "vel_loop_ff_kp" := 10.0;

   // END_IF;

   // // 
   // IF "parameter2" THEN
   //     "model_run" := TRUE;
   //     "controller_run" := TRUE;

   //     "ref_velocity" := 0.0;
   //     "pos_loop_kp" := 0.5;
   //     "pos_loop_Ti" := 0.0;
   //     "vel_loop_kp" := 1.0;
   //     "vel_loop_Ti" := 10.0;
   //     "vel_loop_ff_kp" := 10.0;

   // END_IF;
   // // 
   // IF "parameter3" THEN
   //     "model_run" := TRUE;
   //     "controller_run" := TRUE;

   //     "ref_velocity" := 0.0;
   //     "pos_loop_kp" := 0.5;
   //     "pos_loop_Ti" := 0.0;
   //     "vel_loop_kp" := 1.0;
   //     "vel_loop_Ti" := 10.0;
   //     "vel_loop_ff_kp" := 10.0;

   // END_IF;
   // //
   // IF "parameter4" THEN
   //     "model_run" := TRUE;
   //     "controller_run" := TRUE;

   //     "ref_velocity" := 0.0;
   //     "pos_loop_kp" := 0.5;
   //     "pos_loop_Ti" := 0.0;
   //     "vel_loop_kp" := 1.0;
   //     "vel_loop_Ti" := 10.0;
   //     "vel_loop_ff_kp" := 10.0;

   // END_IF;
   // //
   // IF "parameter5" THEN
   //     "model_run" := TRUE;
   //     "controller_run" := TRUE;

   //     "ref_velocity" := 0.0;
   //     "pos_loop_kp" := 0.5;
   //     "pos_loop_Ti" := 0.0;
   //     "vel_loop_kp" := 1.0;
   //     "vel_loop_Ti" := 10.0;
   //     "vel_loop_ff_kp" := 10.0;

   // END_IF;
END_REGION

REGION Network 14 (SCL): test-14
   // velocity loop
   // IF ("reset0" OR
   //     "reset1" OR
   //     "reset2" OR
   //     "reset3" OR
   //     "reset4")OR
   //     NOT "autotest_run"
   // THEN
   //     "left_cylinder_pos_init" :=1100.0;
   //     "right_cylinder_pos_init" :=900.0;
   //     "ref_velocity" := 0.0;
   //     "model_run" := FALSE;
   //     "controller_run" := FALSE;
   // END_IF;
   // // 
   // IF "parameter1" THEN
   //     "model_run" := TRUE;
   //     "controller_run" := TRUE;

   //     "ref_velocity" := 0.0;
   //     "pos_loop_kp" := 0.5;
   //     "pos_loop_Ti" := 0.0;
   //     "vel_loop_kp" := 1.0;
   //     "vel_loop_Ti" := 10.0;
   //     "vel_loop_ff_kp" := 1.0;

   // END_IF;

   // // 
   // IF "parameter2" THEN
   //     "model_run" := TRUE;
   //     "controller_run" := TRUE;

   //     "ref_velocity" := 0.0;
   //     "pos_loop_kp" := 0.5;
   //     "pos_loop_Ti" := 0.0;
   //     "vel_loop_kp" := 1.0;
   //     "vel_loop_Ti" := 10.0;
   //     "vel_loop_ff_kp" := 10.0;

   // END_IF;
   // // 
   // IF "parameter3" THEN
   //     "model_run" := TRUE;
   //     "controller_run" := TRUE;

   //     "ref_velocity" := 0.0;
   //     "pos_loop_kp" := 0.5;
   //     "pos_loop_Ti" := 0.0;
   //     "vel_loop_kp" := 2.0;
   //     "vel_loop_Ti" := 20.0;
   //     "vel_loop_ff_kp" := 10.0;

   // END_IF;
   // //
   // IF "parameter4" THEN
   //     "model_run" := TRUE;
   //     "controller_run" := TRUE;

   //     "ref_velocity" := 0.0;
   //     "pos_loop_kp" := 0.5;
   //     "pos_loop_Ti" := 0.0;
   //     "vel_loop_kp" := 2.0;
   //     "vel_loop_Ti" := 50.0;
   //     "vel_loop_ff_kp" := 10.0;

   // END_IF;
   // //
   // IF "parameter5" THEN
   //     "model_run" := TRUE;
   //     "controller_run" := TRUE;

   //     "ref_velocity" := 0.0;
   //     "pos_loop_kp" := 0.5;
   //     "pos_loop_Ti" := 0.0;
   //     "vel_loop_kp" := 2.0;
   //     "vel_loop_Ti" := 100.0;
   //     "vel_loop_ff_kp" := 20.0;

   // END_IF;
END_REGION

REGION Network 15 (SCL): test-15
   // velocity loop
   // IF ("reset0" OR
   //     "reset1" OR
   //     "reset2" OR
   //     "reset3" OR
   //     "reset4")OR
   //     NOT "autotest_run"
   // THEN
   //     "left_cylinder_pos_init" :=1100.0;
   //     "right_cylinder_pos_init" :=900.0;
   //     "ref_velocity" := 0.0;
   //     "model_run" := FALSE;
   //     "controller_run" := FALSE;
   // END_IF;
   // // 
   // IF "parameter1" THEN
   //     "model_run" := TRUE;
   //     "controller_run" := TRUE;

   //     "ref_velocity" := 0.0;
   //     "pos_loop_kp" := 0.5;
   //     "pos_loop_Ti" := 0.0;
   //     "vel_loop_kp" := 1.0;
   //     "vel_loop_Ti" := 0.0;
   //     "vel_loop_ff_kp" := 1.0;

   // END_IF;

   // // 
   // IF "parameter2" THEN
   //     "model_run" := TRUE;
   //     "controller_run" := TRUE;

   //     "ref_velocity" := 0.0;
   //     "pos_loop_kp" := 0.5;
   //     "pos_loop_Ti" := 0.0;
   //     "vel_loop_kp" := 2.0;
   //     "vel_loop_Ti" := 0.0;
   //     "vel_loop_ff_kp" := 1.0;

   // END_IF;
   // // 
   // IF "parameter3" THEN
   //     "model_run" := TRUE;
   //     "controller_run" := TRUE;

   //     "ref_velocity" := 0.0;
   //     "pos_loop_kp" := 0.5;
   //     "pos_loop_Ti" := 0.0;
   //     "vel_loop_kp" := 2.0;
   //     "vel_loop_Ti" := 0.0;
   //     "vel_loop_ff_kp" := 10.0;

   // END_IF;
   // //
   // IF "parameter4" THEN
   //     "model_run" := TRUE;
   //     "controller_run" := TRUE;

   //     "ref_velocity" := 0.0;
   //     "pos_loop_kp" := 1;
   //     "pos_loop_Ti" := 0.0;
   //     "vel_loop_kp" := 5.0;
   //     "vel_loop_Ti" := 0.0;
   //     "vel_loop_ff_kp" := 0.0;

   // END_IF;
   // //
   // IF "parameter5" THEN
   //     "model_run" := TRUE;
   //     "controller_run" := TRUE;

   //     "ref_velocity" := 0.0;
   //     "pos_loop_kp" := 0.1;
   //     "pos_loop_Ti" := 0.0;
   //     "vel_loop_kp" := 10.0;
   //     "vel_loop_Ti" := 0.0;
   //     "vel_loop_ff_kp" := 20.0;

   // END_IF;
END_REGION

REGION Network 16 (SCL): test-16
   // velocity loop
   // IF ("reset0" OR
   //     "reset1" OR
   //     "reset2" OR
   //     "reset3" OR
   //     "reset4")OR
   //     NOT "autotest_run"
   // THEN
   //     "left_cylinder_pos_init" :=1000.0;
   //     "right_cylinder_pos_init" :=1000.0;
   //     "ref_velocity" := 0.0;
   //     "model_run" := FALSE;
   //     "controller_run" := FALSE;
   // END_IF;
   // // 
   // IF "parameter1" THEN
   //     "model_run" := TRUE;
   //     "controller_run" := TRUE;

   //     "ref_velocity" := 40.0;
   //     "pos_loop_kp" := 0.5;
   //     "pos_loop_Ti" := 0.0;
   //     "vel_loop_kp" := 1.0;
   //     "vel_loop_Ti" := 0.0;
   //     "vel_loop_ff_kp" := 1.0;

   // END_IF;

   // // 
   // IF "parameter2" THEN
   //     "model_run" := TRUE;
   //     "controller_run" := TRUE;

   //     "ref_velocity" := 40.0;
   //     "pos_loop_kp" := 0.5;
   //     "pos_loop_Ti" := 0.0;
   //     "vel_loop_kp" := 2.0;
   //     "vel_loop_Ti" := 0.0;
   //     "vel_loop_ff_kp" := 1.0;

   // END_IF;
   // // 
   // IF "parameter3" THEN
   //     "model_run" := TRUE;
   //     "controller_run" := TRUE;

   //     "ref_velocity" := 40.0;
   //     "pos_loop_kp" := 0.5;
   //     "pos_loop_Ti" := 0.0;
   //     "vel_loop_kp" := 2.0;
   //     "vel_loop_Ti" := 0.0;
   //     "vel_loop_ff_kp" := 10.0;

   // END_IF;
   // //
   // IF "parameter4" THEN
   //     "model_run" := TRUE;
   //     "controller_run" := TRUE;

   //     "ref_velocity" := 40.0;
   //     "pos_loop_kp" := 1;
   //     "pos_loop_Ti" := 0.0;
   //     "vel_loop_kp" := 5.0;
   //     "vel_loop_Ti" := 0.0;
   //     "vel_loop_ff_kp" := 0.0;

   // END_IF;
   // //
   // IF "parameter5" THEN
   //     "model_run" := TRUE;
   //     "controller_run" := TRUE;

   //     "ref_velocity" := 40.0;
   //     "pos_loop_kp" := 0.1;
   //     "pos_loop_Ti" := 0.0;
   //     "vel_loop_kp" := 10.0;
   //     "vel_loop_Ti" := 0.0;
   //     "vel_loop_ff_kp" := 20.0;

   // END_IF;
END_REGION

REGION Network 17 (SCL): test-17
   // velocity loop
   // IF ("reset0" OR
   //     "reset1" OR
   //     "reset2" OR
   //     "reset3" OR
   //     "reset4")OR
   //     NOT "autotest_run"
   // THEN
   //     "left_cylinder_pos_init" :=1000.0;
   //     "right_cylinder_pos_init" :=1000.0;
   //     "ref_velocity" := 0.0;
   //     "model_run" := FALSE;
   //     "controller_run" := FALSE;
   // END_IF;
   // // 
   // IF "parameter1" THEN
   //     "model_run" := TRUE;
   //     "controller_run" := TRUE;

   //     "ref_velocity" := 40.0;
   //     "pos_loop_kp" := 10.0;
   //     "pos_loop_Ti" := 0.0;
   //     "vel_loop_kp" := 0.0;
   //     "vel_loop_Ti" := 0.0;
   //     "vel_loop_ff_kp" := 1.0;

   // END_IF;

   // // 
   // IF "parameter2" THEN
   //     "model_run" := TRUE;
   //     "controller_run" := TRUE;

   //     "ref_velocity" := 40.0;
   //     "pos_loop_kp" := 0.1;
   //     "pos_loop_Ti" := 0.0;
   //     "vel_loop_kp" := 10.0;
   //     "vel_loop_Ti" := 0.0;
   //     "vel_loop_ff_kp" := 20.0;

   // END_IF;
   // // 
   // IF "parameter3" THEN
   //     "model_run" := TRUE;
   //     "controller_run" := TRUE;

   //     "ref_velocity" := 40.0;
   //     "pos_loop_kp" := 0.1;
   //     "pos_loop_Ti" := 0.0;
   //     "vel_loop_kp" := 10.0;
   //     "vel_loop_Ti" := 100.0;
   //     "vel_loop_ff_kp" := 20.0;

   // END_IF;
   // //
   // IF "parameter4" THEN
   //     "model_run" := TRUE;
   //     "controller_run" := TRUE;

   //     "ref_velocity" := 40.0;
   //     "pos_loop_kp" := 0.5;
   //     "pos_loop_Ti" := 0.0;
   //     "vel_loop_kp" := 5.0;
   //     "vel_loop_Ti" := 100.0;
   //     "vel_loop_ff_kp" := 20.0;

   // END_IF;
   // //
   // IF "parameter5" THEN
   //     "model_run" := TRUE;
   //     "controller_run" := TRUE;

   //     "ref_velocity" := 40.0;
   //     "pos_loop_kp" := 0.5;
   //     "pos_loop_Ti" := 0.0;
   //     "vel_loop_kp" := 5.0;
   //     "vel_loop_Ti" := 50.0;
   //     "vel_loop_ff_kp" := 20.0;

   // END_IF;
END_REGION

REGION Network 18 (SCL): test-18
   // velocity loop
   // IF ("reset0" OR
   //     "reset1" OR
   //     "reset2" OR
   //     "reset3" OR
   //     "reset4")OR
   //     NOT "autotest_run"
   // THEN
   //     "left_cylinder_pos_init" :=1100.0;
   //     "right_cylinder_pos_init" :=900.0;
   //     "ref_velocity" := 0.0;
   //     "model_run" := FALSE;
   //     "controller_run" := FALSE;
   // END_IF;
   // // 
   // IF "parameter1" THEN
   //     "model_run" := TRUE;
   //     "controller_run" := TRUE;

   //     "ref_velocity" := 0.0;
   //     "pos_loop_kp" := 10.0;
   //     "pos_loop_Ti" := 0.0;
   //     "vel_loop_kp" := 0.0;
   //     "vel_loop_Ti" := 0.0;
   //     "vel_loop_ff_kp" := 1.0;

   // END_IF;

   // // 
   // IF "parameter2" THEN
   //     "model_run" := TRUE;
   //     "controller_run" := TRUE;

   //     "ref_velocity" := 0.0;
   //     "pos_loop_kp" := 0.1;
   //     "pos_loop_Ti" := 0.0;
   //     "vel_loop_kp" := 10.0;
   //     "vel_loop_Ti" := 0.0;
   //     "vel_loop_ff_kp" := 20.0;

   // END_IF;
   // // 
   // IF "parameter3" THEN
   //     "model_run" := TRUE;
   //     "controller_run" := TRUE;

   //     "ref_velocity" := 0.0;
   //     "pos_loop_kp" := 0.1;
   //     "pos_loop_Ti" := 0.0;
   //     "vel_loop_kp" := 10.0;
   //     "vel_loop_Ti" := 100.0;
   //     "vel_loop_ff_kp" := 20.0;

   // END_IF;
   // //
   // IF "parameter4" THEN
   //     "model_run" := TRUE;
   //     "controller_run" := TRUE;

   //     "ref_velocity" := 0.0;
   //     "pos_loop_kp" := 0.5;
   //     "pos_loop_Ti" := 0.0;
   //     "vel_loop_kp" := 5.0;
   //     "vel_loop_Ti" := 100.0;
   //     "vel_loop_ff_kp" := 20.0;

   // END_IF;
   // //
   // IF "parameter5" THEN
   //     "model_run" := TRUE;
   //     "controller_run" := TRUE;

   //     "ref_velocity" := 0.0;
   //     "pos_loop_kp" := 0.5;
   //     "pos_loop_Ti" := 0.0;
   //     "vel_loop_kp" := 5.0;
   //     "vel_loop_Ti" := 50.0;
   //     "vel_loop_ff_kp" := 20.0;

   // END_IF;
END_REGION

REGION Network 19 (SCL): test-19
   // velocity loop
   // IF ("reset0" OR
   //     "reset1" OR
   //     "reset2" OR
   //     "reset3" OR
   //     "reset4")OR
   //     NOT "autotest_run"
   // THEN
   //     "left_cylinder_pos_init" :=1000.0;
   //     "right_cylinder_pos_init" :=1000.0;
   //     "ref_velocity" := 0.0;
   //     "model_run" := FALSE;
   //     "controller_run" := FALSE;
   // END_IF;
   // // 
   // IF "parameter1" THEN
   //     "model_run" := TRUE;
   //     "controller_run" := TRUE;

   //     "ref_velocity" := 40.0;
   //     "pos_loop_kp" := 10.0;
   //     "pos_loop_Ti" := 0.0;
   //     "vel_loop_kp" := 0.0;
   //     "vel_loop_Ti" := 0.0;
   //     "vel_loop_ff_kp" := 1.0;

   // END_IF;

   // // 
   // IF "parameter2" THEN
   //     "model_run" := TRUE;
   //     "controller_run" := TRUE;

   //     "ref_velocity" := 40.0;
   //     "pos_loop_kp" := 0.1;
   //     "pos_loop_Ti" := 0.0;
   //     "vel_loop_kp" := 10.0;
   //     "vel_loop_Ti" := 0.0;
   //     "vel_loop_ff_kp" := 0.0;

   // END_IF;
   // // 
   // IF "parameter3" THEN
   //     "model_run" := TRUE;
   //     "controller_run" := TRUE;

   //     "ref_velocity" := 40.0;
   //     "pos_loop_kp" := 0.1;
   //     "pos_loop_Ti" := 0.0;
   //     "vel_loop_kp" := 10.0;
   //     "vel_loop_Ti" := 0.0;
   //     "vel_loop_ff_kp" := 10.0;

   // END_IF;
   // //
   // IF "parameter4" THEN
   //     "model_run" := TRUE;
   //     "controller_run" := TRUE;

   //     "ref_velocity" := 40.0;
   //     "pos_loop_kp" := 0.1;
   //     "pos_loop_Ti" := 0.0;
   //     "vel_loop_kp" := 10.0;
   //     "vel_loop_Ti" := 0.0;
   //     "vel_loop_ff_kp" := 50.0;

   // END_IF;
   // //
   // IF "parameter5" THEN
   //     "model_run" := TRUE;
   //     "controller_run" := TRUE;

   //     "ref_velocity" := 40.0;
   //     "pos_loop_kp" := 0.1;
   //     "pos_loop_Ti" := 0.0;
   //     "vel_loop_kp" := 10.0;
   //     "vel_loop_Ti" := 0.0;
   //     "vel_loop_ff_kp" := 100.0;

   // END_IF;
END_REGION

REGION Network 20 (SCL): test-20
   // velocity loop
   // IF ("reset0" OR
   //     "reset1" OR
   //     "reset2" OR
   //     "reset3" OR
   //     "reset4")OR
   //     NOT "autotest_run"
   // THEN
   //     "left_cylinder_pos_init" :=1000.0;
   //     "right_cylinder_pos_init" :=1000.0;
   //     "ref_velocity" := 0.0;
   //     "model_run" := FALSE;
   //     "controller_run" := FALSE;
   // END_IF;
   // // 
   // IF "parameter1" THEN
   //     "model_run" := TRUE;
   //     "controller_run" := TRUE;

   //     "ref_velocity" := 40.0;
   //     "pos_loop_kp" := 1.0;
   //     "pos_loop_Ti" := 0.0;
   //     "vel_loop_kp" := 0.0;
   //     "vel_loop_Ti" := 0.0;
   //     "vel_loop_ff_kp" := 1.0;

   // END_IF;

   // // 
   // IF "parameter2" THEN
   //     "model_run" := TRUE;
   //     "controller_run" := TRUE;

   //     "ref_velocity" := 40.0;
   //     "pos_loop_kp" := 0.1;
   //     "pos_loop_Ti" := 0.0;
   //     "vel_loop_kp" := 10.0;
   //     "vel_loop_Ti" := 0.0;
   //     "vel_loop_ff_kp" := 100.0;

   // END_IF;
   // // 
   // IF "parameter3" THEN
   //     "model_run" := TRUE;
   //     "controller_run" := TRUE;

   //     "ref_velocity" := 40.0;
   //     "pos_loop_kp" := 0.1;
   //     "pos_loop_Ti" := 0.0;
   //     "vel_loop_kp" := 5.0;
   //     "vel_loop_Ti" := 0.0;
   //     "vel_loop_ff_kp" := 100.0;

   // END_IF;
   // //
   // IF "parameter4" THEN
   //     "model_run" := TRUE;
   //     "controller_run" := TRUE;

   //     "ref_velocity" := 40.0;
   //     "pos_loop_kp" := 0.1;
   //     "pos_loop_Ti" := 0.0;
   //     "vel_loop_kp" := 5.0;
   //     "vel_loop_Ti" := 100.0;
   //     "vel_loop_ff_kp" := 100.0;

   // END_IF;
   // //
   // IF "parameter5" THEN
   //     "model_run" := TRUE;
   //     "controller_run" := TRUE;

   //     "ref_velocity" := 40.0;
   //     "pos_loop_kp" := 0.1;
   //     "pos_loop_Ti" := 0.0;
   //     "vel_loop_kp" := 5.0;
   //     "vel_loop_Ti" := 500.0;
   //     "vel_loop_ff_kp" := 100.0;

   // END_IF;
END_REGION

REGION Network 21 (SCL): test-20
   // velocity loop
   // IF ("reset0" OR
   //     "reset1" OR
   //     "reset2" OR
   //     "reset3" OR
   //     "reset4")OR
   //     NOT "autotest_run"
   // THEN
   //     "left_cylinder_pos_init" :=1100.0;
   //     "right_cylinder_pos_init" :=900.0;
   //     "ref_velocity" := 0.0;
   //     "model_run" := FALSE;
   //     "controller_run" := FALSE;
   // END_IF;
   // // 
   // IF "parameter1" THEN
   //     "model_run" := TRUE;
   //     "controller_run" := TRUE;

   //     "ref_velocity" := 0.0;
   //     "pos_loop_kp" := 10.0;
   //     "pos_loop_Ti" := 0.0;
   //     "vel_loop_kp" := 0.0;
   //     "vel_loop_Ti" := 0.0;
   //     "vel_loop_ff_kp" := 1.0;

   // END_IF;

   // // 
   // IF "parameter2" THEN
   //     "model_run" := TRUE;
   //     "controller_run" := TRUE;

   //     "ref_velocity" := 0.0;
   //     "pos_loop_kp" := 0.1;
   //     "pos_loop_Ti" := 0.0;
   //     "vel_loop_kp" := 10.0;
   //     "vel_loop_Ti" := 0.0;
   //     "vel_loop_ff_kp" := 100.0;

   // END_IF;
   // // 
   // IF "parameter3" THEN
   //     "model_run" := TRUE;
   //     "controller_run" := TRUE;

   //     "ref_velocity" := 0.0;
   //     "pos_loop_kp" := 0.1;
   //     "pos_loop_Ti" := 0.0;
   //     "vel_loop_kp" := 5.0;
   //     "vel_loop_Ti" := 0.0;
   //     "vel_loop_ff_kp" := 100.0;

   // END_IF;
   // //
   // IF "parameter4" THEN
   //     "model_run" := TRUE;
   //     "controller_run" := TRUE;

   //     "ref_velocity" := 0.0;
   //     "pos_loop_kp" := 0.1;
   //     "pos_loop_Ti" := 0.0;
   //     "vel_loop_kp" := 5.0;
   //     "vel_loop_Ti" := 1000.0;
   //     "vel_loop_ff_kp" := 100.0;

   // END_IF;
   // //
   // IF "parameter5" THEN
   //     "model_run" := TRUE;
   //     "controller_run" := TRUE;

   //     "ref_velocity" := 0.0;
   //     "pos_loop_kp" := 0.1;
   //     "pos_loop_Ti" := 0.0;
   //     "vel_loop_kp" := 10.0;
   //     "vel_loop_Ti" := 5000.0;
   //     "vel_loop_ff_kp" := 100.0;

   // END_IF;
END_REGION

REGION Network 22 (SCL): recommandation
   // velocity loop
   // IF ("reset0" OR
   //     "reset1" OR
   //     "reset2" OR
   //     "reset3" OR
   //     "reset4")OR
   //     NOT "autotest_run"
   // THEN
   //     "left_cylinder_pos_init" :=1100.0;
   //     "right_cylinder_pos_init" :=900.0;
   //     "ref_velocity" := 0.0;
   //     "model_run" := FALSE;
   //     "controller_run" := FALSE;
   // END_IF;
   // // 
   // IF "parameter1" THEN
   //     "model_run" := TRUE;
   //     "controller_run" := TRUE;

   //     "ref_velocity" := 0.0;
   //     "pos_loop_kp" := 10.0;
   //     "pos_loop_Ti" := 0.0;
   //     "vel_loop_kp" := 0.0;
   //     "vel_loop_Ti" := 0.0;
   //     "vel_loop_ff_kp" := 1.0;

   // END_IF;

   // // best parameter
   // IF "parameter2" THEN
   //     "model_run" := TRUE;
   //     "controller_run" := TRUE;

   //     "ref_velocity" := 40.0;
   //     "pos_loop_kp" := 0.1;
   //     "pos_loop_Ti" := 0.0;
   //     "vel_loop_kp" := 10.0;
   //     "vel_loop_Ti" := 0.0;
   //     "vel_loop_ff_kp" := 100.0;

   // END_IF;
   // // 
   // IF "parameter3" THEN
   //     "model_run" := TRUE;
   //     "controller_run" := TRUE;

   //     "ref_velocity" := 40.0;
   //     "pos_loop_kp" := 0.1;
   //     "pos_loop_Ti" := 0.0;
   //     "vel_loop_kp" := 5.0;
   //     "vel_loop_Ti" := 0.0;
   //     "vel_loop_ff_kp" := 100.0;

   // END_IF;
   // //
   // IF "parameter4" THEN
   //     "model_run" := TRUE;
   //     "controller_run" := TRUE;

   //     "ref_velocity" := 40.0;
   //     "pos_loop_kp" := 0.1;
   //     "pos_loop_Ti" := 0.0;
   //     "vel_loop_kp" := 5.0;
   //     "vel_loop_Ti" := 1000.0;
   //     "vel_loop_ff_kp" := 100.0;

   // END_IF;
   // //
   // IF "parameter5" THEN
   //     "model_run" := TRUE;
   //     "controller_run" := TRUE;

   //     "ref_velocity" := 40.0;
   //     "pos_loop_kp" := 0.1;
   //     "pos_loop_Ti" := 0.0;
   //     "vel_loop_kp" := 10.0;
   //     "vel_loop_Ti" := 5000.0;
   //     "vel_loop_ff_kp" := 100.0;

   // END_IF;
END_REGION

REGION Network 23 (SCL): 4 Paper-1
   // velocity loop
   // IF ("reset0" OR
   //     "reset1" OR
   //     "reset2" OR
   //     "reset3" OR
   //     "reset4")OR
   //     NOT "autotest_run"
   // THEN
   //     "left_cylinder_pos_init" :=1100.0;
   //     "right_cylinder_pos_init" :=900.0;
   //     "ref_velocity" := 0.0;
   //     "model_run" := FALSE;
   //     "controller_run" := FALSE;
   // END_IF;
   // // 
   // IF "parameter1" THEN
   //     "model_run" := TRUE;
   //     "controller_run" := TRUE;

   //     "ref_velocity" := 0.0;
   //     "pos_loop_kp" := 1.0;
   //     "pos_loop_Ti" := 0.0;
   //     "vel_loop_kp" := 0.0;
   //     "vel_loop_Ti" := 0.0;
   //     "vel_loop_ff_kp" := 1.0;

   // END_IF;

   // // best parameter
   // IF "parameter2" THEN
   //     "model_run" := TRUE;
   //     "controller_run" := TRUE;

   //     "ref_velocity" := 0.0;
   //     "pos_loop_kp" := 10.0;
   //     "pos_loop_Ti" := 0.0;
   //     "vel_loop_kp" := 0.0;
   //     "vel_loop_Ti" := 0.0;
   //     "vel_loop_ff_kp" := 1.0;

   // END_IF;
   // // 
   // IF "parameter3" THEN
   //     "model_run" := TRUE;
   //     "controller_run" := TRUE;

   //     "ref_velocity" := 0.0;
   //     "pos_loop_kp" := 30.0;
   //     "pos_loop_Ti" := 0.0;
   //     "vel_loop_kp" := 0.0;
   //     "vel_loop_Ti" := 0.0;
   //     "vel_loop_ff_kp" := 1.0;

   // END_IF;
   // //
   // IF "parameter4" THEN
   //     "model_run" := TRUE;
   //     "controller_run" := TRUE;

   //     "ref_velocity" := 0.0;
   //     "pos_loop_kp" := 50.0;
   //     "pos_loop_Ti" := 0.0;
   //     "vel_loop_kp" := 0.0;
   //     "vel_loop_Ti" := 0.0;
   //     "vel_loop_ff_kp" := 1.0;

   // END_IF;
   // //
   // IF "parameter5" THEN
   //     "model_run" := TRUE;
   //     "controller_run" := TRUE;

   //     "ref_velocity" := 0.0;
   //     "pos_loop_kp" := 100.0;
   //     "pos_loop_Ti" := 0.0;
   //     "vel_loop_kp" := 0.0;
   //     "vel_loop_Ti" := 0.0;
   //     "vel_loop_ff_kp" := 1.0;

   // END_IF;
END_REGION

REGION Network 24 (SCL): 4 Paper-2
   // velocity loop
   // IF ("reset0" OR
   //     "reset1" OR
   //     "reset2" OR
   //     "reset3" OR
   //     "reset4")OR
   //     NOT "autotest_run"
   // THEN
   //     "left_cylinder_pos_init" :=1000.0;
   //     "right_cylinder_pos_init" :=1000.0;
   //     "ref_velocity" := 0.0;
   //     "model_run" := FALSE;
   //     "controller_run" := FALSE;
   // END_IF;
   // // 
   // IF "parameter1" THEN
   //     "model_run" := TRUE;
   //     "controller_run" := TRUE;

   //     "ref_velocity" := 40.0;
   //     "pos_loop_kp" := 1.0;
   //     "pos_loop_Ti" := 0.0;
   //     "vel_loop_kp" := 0.0;
   //     "vel_loop_Ti" := 0.0;
   //     "vel_loop_ff_kp" := 1.0;

   // END_IF;

   // // best parameter
   // IF "parameter2" THEN
   //     "model_run" := TRUE;
   //     "controller_run" := TRUE;

   //     "ref_velocity" := 40.0;
   //     "pos_loop_kp" := 10.0;
   //     "pos_loop_Ti" := 0.0;
   //     "vel_loop_kp" := 0.0;
   //     "vel_loop_Ti" := 0.0;
   //     "vel_loop_ff_kp" := 1.0;

   // END_IF;
   // // 
   // IF "parameter3" THEN
   //     "model_run" := TRUE;
   //     "controller_run" := TRUE;

   //     "ref_velocity" := 40.0;
   //     "pos_loop_kp" := 30.0;
   //     "pos_loop_Ti" := 0.0;
   //     "vel_loop_kp" := 0.0;
   //     "vel_loop_Ti" := 0.0;
   //     "vel_loop_ff_kp" := 1.0;

   // END_IF;
   // //
   // IF "parameter4" THEN
   //     "model_run" := TRUE;
   //     "controller_run" := TRUE;

   //     "ref_velocity" := 40.0;
   //     "pos_loop_kp" := 50.0;
   //     "pos_loop_Ti" := 0.0;
   //     "vel_loop_kp" := 0.0;
   //     "vel_loop_Ti" := 0.0;
   //     "vel_loop_ff_kp" := 1.0;

   // END_IF;
   // //
   // IF "parameter5" THEN
   //     "model_run" := TRUE;
   //     "controller_run" := TRUE;

   //     "ref_velocity" := 40.0;
   //     "pos_loop_kp" := 100.0;
   //     "pos_loop_Ti" := 0.0;
   //     "vel_loop_kp" := 0.0;
   //     "vel_loop_Ti" := 0.0;
   //     "vel_loop_ff_kp" := 1.0;

   // END_IF;
END_REGION

REGION Network 25 (SCL): 4 Paper-3
   // velocity loop
   // IF ("reset0" OR
   //     "reset1" OR
   //     "reset2" OR
   //     "reset3" OR
   //     "reset4")OR
   //     NOT "autotest_run"
   // THEN
   //     "left_cylinder_pos_init" := 1000.0;
   //     "right_cylinder_pos_init" := 1000.0;
   //     "ref_velocity" := 0.0;
   //     "model_run" := FALSE;
   //     "controller_run" := FALSE;
   // END_IF;
   // // 
   // IF "parameter1" THEN
   //     "model_run" := TRUE;
   //     "controller_run" := TRUE;

   //     "ref_velocity" := 40.0;
   //     "pos_loop_kp" := 1.0;
   //     "pos_loop_Ti" := 0.0;
   //     "vel_loop_kp" := 1.0;
   //     "vel_loop_Ti" := 0.0;
   //     "vel_loop_ff_kp" := 0.0;

   // END_IF;

   // // best parameter
   // IF "parameter2" THEN
   //     "model_run" := TRUE;
   //     "controller_run" := TRUE;

   //     "ref_velocity" := 40.0;
   //     "pos_loop_kp" := 1.0;
   //     "pos_loop_Ti" := 0.0;
   //     "vel_loop_kp" := 10.0;
   //     "vel_loop_Ti" := 0.0;
   //     "vel_loop_ff_kp" := 0.0;

   // END_IF;
   // // 
   // IF "parameter3" THEN
   //     "model_run" := TRUE;
   //     "controller_run" := TRUE;

   //     "ref_velocity" := 40.0;
   //     "pos_loop_kp" := 1.0;
   //     "pos_loop_Ti" := 0.0;
   //     "vel_loop_kp" := 20.0;
   //     "vel_loop_Ti" := 0.0;
   //     "vel_loop_ff_kp" := 0.0;

   // END_IF;
   // //
   // IF "parameter4" THEN
   //     "model_run" := TRUE;
   //     "controller_run" := TRUE;

   //     "ref_velocity" := 40.0;
   //     "pos_loop_kp" := 0.1;
   //     "pos_loop_Ti" := 0.0;
   //     "vel_loop_kp" := 10.0;
   //     "vel_loop_Ti" := 0.0;
   //     "vel_loop_ff_kp" := 0.0;

   // END_IF;
   // //
   // IF "parameter5" THEN
   //     "model_run" := TRUE;
   //     "controller_run" := TRUE;

   //     "ref_velocity" := 40.0;
   //     "pos_loop_kp" := 0.1;
   //     "pos_loop_Ti" := 0.0;
   //     "vel_loop_kp" := 20.0;
   //     "vel_loop_Ti" := 0.0;
   //     "vel_loop_ff_kp" := 0.0;

   // END_IF;
END_REGION

REGION Network 26 (SCL): 4 Paper-4
   // velocity loop
   // IF ("reset0" OR
   //     "reset1" OR
   //     "reset2" OR
   //     "reset3" OR
   //     "reset4")OR
   //     NOT "autotest_run"
   // THEN
   //     "left_cylinder_pos_init" := 1100.0;
   //     "right_cylinder_pos_init" := 900.0;
   //     "ref_velocity" := 0.0;
   //     "model_run" := FALSE;
   //     "controller_run" := FALSE;
   // END_IF;
   // // 
   // IF "parameter1" THEN
   //     "model_run" := TRUE;
   //     "controller_run" := TRUE;

   //     "ref_velocity" := 0.0;
   //     "pos_loop_kp" := 1.0;
   //     "pos_loop_Ti" := 0.0;
   //     "vel_loop_kp" := 1.0;
   //     "vel_loop_Ti" := 0.0;
   //     "vel_loop_ff_kp" := 0.0;

   // END_IF;

   // // best parameter
   // IF "parameter2" THEN
   //     "model_run" := TRUE;
   //     "controller_run" := TRUE;

   //     "ref_velocity" := 0.0;
   //     "pos_loop_kp" := 1.0;
   //     "pos_loop_Ti" := 0.0;
   //     "vel_loop_kp" := 10.0;
   //     "vel_loop_Ti" := 0.0;
   //     "vel_loop_ff_kp" := 0.0;

   // END_IF;
   // // 
   // IF "parameter3" THEN
   //     "model_run" := TRUE;
   //     "controller_run" := TRUE;

   //     "ref_velocity" := 0.0;
   //     "pos_loop_kp" := 1.0;
   //     "pos_loop_Ti" := 0.0;
   //     "vel_loop_kp" := 20.0;
   //     "vel_loop_Ti" := 0.0;
   //     "vel_loop_ff_kp" := 0.0;

   // END_IF;
   // //
   // IF "parameter4" THEN
   //     "model_run" := TRUE;
   //     "controller_run" := TRUE;

   //     "ref_velocity" := 0.0;
   //     "pos_loop_kp" := 0.1;
   //     "pos_loop_Ti" := 0.0;
   //     "vel_loop_kp" := 10.0;
   //     "vel_loop_Ti" := 0.0;
   //     "vel_loop_ff_kp" := 0.0;

   // END_IF;
   // //
   // IF "parameter5" THEN
   //     "model_run" := TRUE;
   //     "controller_run" := TRUE;

   //     "ref_velocity" := 0.0;
   //     "pos_loop_kp" := 0.1;
   //     "pos_loop_Ti" := 0.0;
   //     "vel_loop_kp" := 20.0;
   //     "vel_loop_Ti" := 0.0;
   //     "vel_loop_ff_kp" := 0.0;

   // END_IF;
END_REGION

REGION Network 27 (SCL): 4 Paper-5-1
   // velocity loop
   // IF ("reset0" OR
   //     "reset1" OR
   //     "reset2" OR
   //     "reset3" OR
   //     "reset4")OR
   //     NOT "autotest_run"
   // THEN
   //     "left_cylinder_pos_init" := 1100.0;
   //     "right_cylinder_pos_init" := 900.0;
   //     "ref_velocity" := 0.0;
   //     "model_run" := FALSE;
   //     "controller_run" := FALSE;
   // END_IF;
   // // 
   // IF "parameter1" THEN
   //     "model_run" := TRUE;
   //     "controller_run" := TRUE;

   //     "ref_velocity" := 0.0;
   //     "pos_loop_kp" := 0.1;
   //     "pos_loop_Ti" := 0.0;
   //     "vel_loop_kp" := 10.0;
   //     "vel_loop_Ti" := 0.0;
   //     "vel_loop_ff_kp" := 100.0;

   // END_IF;

   // // best parameter
   // IF "parameter2" THEN
   //     "model_run" := TRUE;
   //     "controller_run" := TRUE;

   //     "ref_velocity" := 40.0;
   //     "pos_loop_kp" := 0.1;
   //     "pos_loop_Ti" := 0.0;
   //     "vel_loop_kp" := 10.0;
   //     "vel_loop_Ti" := 0.0;
   //     "vel_loop_ff_kp" := 100.0;

   // END_IF;
   // // 
   // IF "parameter3" THEN
   //     "model_run" := TRUE;
   //     "controller_run" := TRUE;

   //     "ref_velocity" := 0.0;
   //     "pos_loop_kp" := 0.0;
   //     "pos_loop_Ti" := 0.0;
   //     "vel_loop_kp" := 0.0;
   //     "vel_loop_Ti" := 0.0;
   //     "vel_loop_ff_kp" := 0.0;

   // END_IF;
   // //
   // IF "parameter4" THEN
   //     "model_run" := TRUE;
   //     "controller_run" := TRUE;

   //     "ref_velocity" := 0.0;
   //     "pos_loop_kp" := 0.0;
   //     "pos_loop_Ti" := 0.0;
   //     "vel_loop_kp" := 0.0;
   //     "vel_loop_Ti" := 0.0;
   //     "vel_loop_ff_kp" := 0.0;

   // END_IF;
   // //
   // IF "parameter5" THEN
   //     "model_run" := TRUE;
   //     "controller_run" := TRUE;

   //     "ref_velocity" := 0.0;
   //     "pos_loop_kp" := 0.0;
   //     "pos_loop_Ti" := 0.0;
   //     "vel_loop_kp" := 0.0;
   //     "vel_loop_Ti" := 0.0;
   //     "vel_loop_ff_kp" := 0.0;

   // END_IF;
END_REGION

REGION Network 28 (SCL): 4 Paper-5-2
   // velocity loop
   IF ("reset0" OR
       "reset1" OR
       "reset2" OR
       "reset3" OR
       "reset4") OR
       NOT "autotest_run"
   THEN
       "left_cylinder_pos_init" := 1100.0;
       "right_cylinder_pos_init" := 900.0;
       "ref_velocity" := 0.0;
       "model_run" := FALSE;
       "controller_run" := FALSE;
   END_IF;
   // 
   IF "parameter1" THEN
       "model_run" := TRUE;
       "controller_run" := TRUE;

       "ref_velocity" := 40.0;
       "pos_loop_kp" := 0.1;
       "pos_loop_Ti" := 0.0;
       "vel_loop_kp" := 10.0;
       "vel_loop_Ti" := 10.0;
       "vel_loop_ff_kp" := 100.0;

   END_IF;

   // best parameter
   IF "parameter2" THEN
       "model_run" := TRUE;
       "controller_run" := TRUE;

       "ref_velocity" := 40.0;
       "pos_loop_kp" := 0.1;
       "pos_loop_Ti" := 0.0;
       "vel_loop_kp" := 10.0;
       "vel_loop_Ti" := 0.0;
       "vel_loop_ff_kp" := 100.0;

   END_IF;
   // 
   IF "parameter3" THEN
       "model_run" := TRUE;
       "controller_run" := TRUE;

       "ref_velocity" := 0.0;
       "pos_loop_kp" := 0.0;
       "pos_loop_Ti" := 0.0;
       "vel_loop_kp" := 0.0;
       "vel_loop_Ti" := 0.0;
       "vel_loop_ff_kp" := 0.0;

   END_IF;
   //
   IF "parameter4" THEN
       "model_run" := TRUE;
       "controller_run" := TRUE;

       "ref_velocity" := 0.0;
       "pos_loop_kp" := 0.0;
       "pos_loop_Ti" := 0.0;
       "vel_loop_kp" := 0.0;
       "vel_loop_Ti" := 0.0;
       "vel_loop_ff_kp" := 0.0;

   END_IF;
   //
   IF "parameter5" THEN
       "model_run" := TRUE;
       "controller_run" := TRUE;

       "ref_velocity" := 0.0;
       "pos_loop_kp" := 0.0;
       "pos_loop_Ti" := 0.0;
       "vel_loop_kp" := 0.0;
       "vel_loop_Ti" := 0.0;
       "vel_loop_ff_kp" := 0.0;

   END_IF;
END_REGION
END_ORGANIZATION_BLOCK

// folder: ctrl_synch/controller

FUNCTION_BLOCK "controller"   // FB7, LAD
{ S7_Optimized_Access := 'TRUE' }
VERSION : 0.1
   VAR_INPUT
      run : Bool;
      ref_velocity : Real;
      ref_vel_ramp_acc : Real;
      ref_vel_min : Real;
      ref_vel_max : Real;
      left_pos : Real;
      left_pos_tau : Real;
      "left_vel_fb%" : Real;
      right_pos : Real;
      right_pos_tau : Real;
      "right_vel_fb%" : Real;
      pos_loop_dbw : Real;
      pos_loop_kp : Real;
      "pos_loop_Ti[s]" : Real;
      pos_loop_min : Real;
      pos_loop_max : Real;
      vel_loop_dbw : Real;
      vel_loop_kp : Real;
      "vel_loop_Ti[s]" : Real;
      vel_loop_ff_kp : Real;
      vel_loop_min : Real;
      vel_loop_max : Real;
      "cycle[s]" : Real;
   END_VAR
   VAR_OUTPUT
      ref_vel_add : Real;
      left_vel_cmd : Real;
      right_vel_cmd : Real;
      left_pos_cmd : Real;
      right_pos_cmd : Real;
      left_vel_fb : Real;
      right_vel_fb : Real;
   END_VAR
   VAR
      ref_vel_ramp : Real;
      LAG1_Instance_left_pos : "LAG1";
      LAG1_Instance_right_pos : "LAG1";
      DERIVATIVE_Instance_left_vel : "DERIVATIVE";
      DERIVATIVE_Instance_right_vel : "DERIVATIVE";
      pos_loop_Instance_left : "pos_loop";
      vel_loop_Instance_left : "vel_loop";
      pos_loop_Instance_right : "pos_loop";
      vel_loop_Instance_right : "vel_loop";
   END_VAR
   VAR_TEMP
      left_pos_fb : Real;
      right_pos_fb : Real;
      left_vel_lowpass_out : Real;
      right_vel_lowpass_out : Real;
      cycle_ms : Real;
      B_ParamErr : Bool;
      B_EndRmp : Bool;
      B_ZeroRmp : Bool;
      B_Acc : Bool;
      B_Dec : Bool;
      R_Acc : Real;
      ref_pos : Real;
      vel_fb : Real;
   END_VAR
   VAR_TEMP   // added for the SCL form of the ladder/FBD networks
      _w1 : Bool;
   END_VAR
BEGIN

REGION Network 1
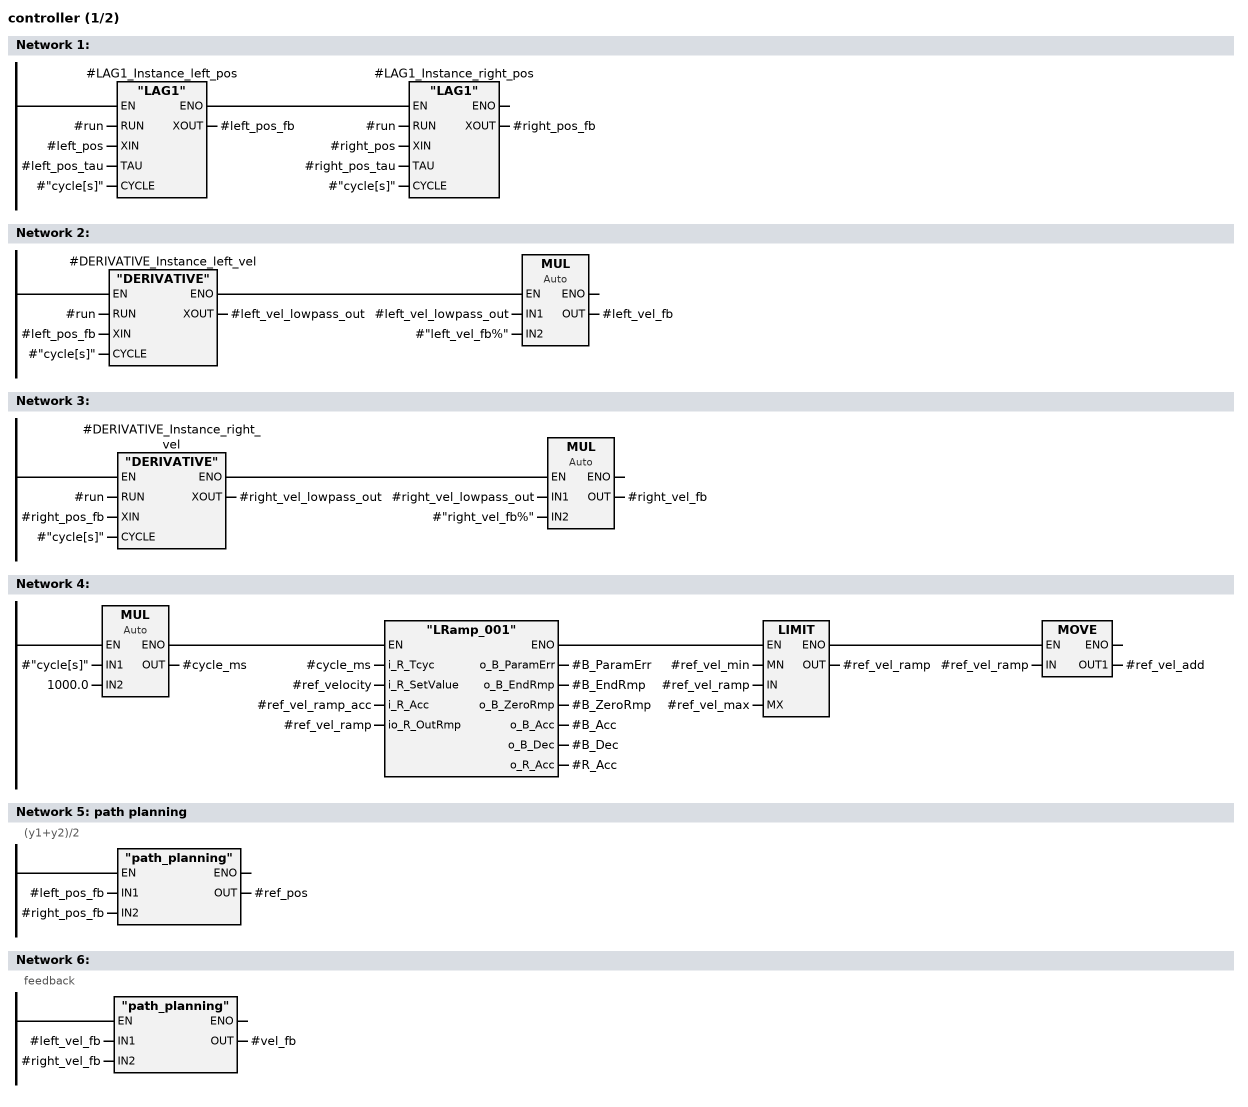
   RUNG wire#powerrail
      #LAG1_Instance_left_pos(RUN := #run, XIN := #left_pos, TAU := #left_pos_tau, CYCLE := #"cycle[s]", XOUT => #left_pos_fb)
      #LAG1_Instance_right_pos(RUN := #run, XIN := #right_pos, TAU := #right_pos_tau, CYCLE := #"cycle[s]", XOUT => #right_pos_fb)
   END_RUNG
   // the same network as SCL:
   #LAG1_Instance_left_pos(RUN := #run,   // "LAG1"
                           XIN := #left_pos,
                           TAU := #left_pos_tau,
                           CYCLE := #"cycle[s]",
                           XOUT => #left_pos_fb,
                           ENO => #_w1);
   IF #_w1 THEN
       #LAG1_Instance_right_pos(RUN := #run,   // "LAG1"
                               XIN := #right_pos,
                               TAU := #right_pos_tau,
                               CYCLE := #"cycle[s]",
                               XOUT => #right_pos_fb);
   END_IF;
END_REGION

REGION Network 2
   RUNG wire#powerrail
      #DERIVATIVE_Instance_left_vel(RUN := #run, XIN := #left_pos_fb, CYCLE := #"cycle[s]", XOUT => #left_vel_lowpass_out)
      Mul(in1 := #left_vel_lowpass_out, in2 := #"left_vel_fb%", out => #left_vel_fb)
   END_RUNG
   // the same network as SCL:
   #DERIVATIVE_Instance_left_vel(RUN := #run,   // "DERIVATIVE"
                           XIN := #left_pos_fb,
                           CYCLE := #"cycle[s]",
                           XOUT => #left_vel_lowpass_out,
                           ENO => #_w1);
   IF #_w1 THEN #left_vel_fb := #left_vel_lowpass_out * #"left_vel_fb%"; END_IF;
END_REGION

REGION Network 3
   RUNG wire#powerrail
      #DERIVATIVE_Instance_right_vel(RUN := #run, XIN := #right_pos_fb, CYCLE := #"cycle[s]", XOUT => #right_vel_lowpass_out)
      Mul(in1 := #right_vel_lowpass_out, in2 := #"right_vel_fb%", out => #right_vel_fb)
   END_RUNG
   // the same network as SCL:
   #DERIVATIVE_Instance_right_vel(RUN := #run,   // "DERIVATIVE"
                           XIN := #right_pos_fb,
                           CYCLE := #"cycle[s]",
                           XOUT => #right_vel_lowpass_out,
                           ENO => #_w1);
   IF #_w1 THEN #right_vel_fb := #right_vel_lowpass_out * #"right_vel_fb%"; END_IF;
END_REGION

REGION Network 4
   #cycle_ms := #"cycle[s]" * 1000.0;
   "LRamp_001"(i_R_Tcyc := #cycle_ms,
               i_R_SetValue := #ref_velocity,
               i_R_Acc := #ref_vel_ramp_acc,
               io_R_OutRmp := #ref_vel_ramp,
               o_B_ParamErr => #B_ParamErr,
               o_B_EndRmp => #B_EndRmp,
               o_B_ZeroRmp => #B_ZeroRmp,
               o_B_Acc => #B_Acc,
               o_B_Dec => #B_Dec,
               o_R_Acc => #R_Acc,
               ENO => #_w1);
   IF #_w1 THEN
       #ref_vel_ramp := LIMIT(MN := #ref_vel_min, IN := #ref_vel_ramp, MX := #ref_vel_max);
       #ref_vel_add := #ref_vel_ramp;
   END_IF;
END_REGION

REGION Network 5: path planning
   // (y1+y2)/2
   RUNG wire#powerrail
      "path_planning"(IN1 := #left_pos_fb, IN2 := #right_pos_fb, OUT => #ref_pos)
   END_RUNG
   // the same network as SCL:
   "path_planning"(IN1 := #left_pos_fb, IN2 := #right_pos_fb, OUT => #ref_pos);
END_REGION

REGION Network 6
   // feedback
   RUNG wire#powerrail
      "path_planning"(IN1 := #left_vel_fb, IN2 := #right_vel_fb, OUT => #vel_fb)
   END_RUNG
   // the same network as SCL:
   "path_planning"(IN1 := #left_vel_fb, IN2 := #right_vel_fb, OUT => #vel_fb);
END_REGION

REGION Network 7
   // feedback
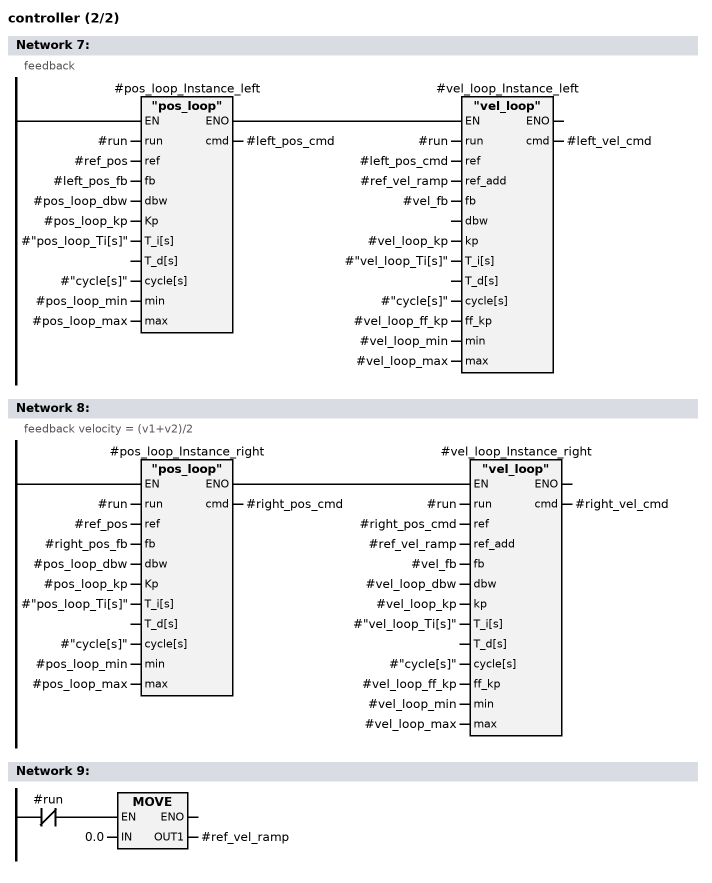
   RUNG wire#powerrail
      #pos_loop_Instance_left(run := #run, ref := #ref_pos, fb := #left_pos_fb, dbw := #pos_loop_dbw, Kp := #pos_loop_kp, "T_i[s]" := #"pos_loop_Ti[s]", "T_d[s]" :=, "cycle[s]" := #"cycle[s]", min := #pos_loop_min, max := #pos_loop_max, cmd => #left_pos_cmd)
      #vel_loop_Instance_left(run := #run, ref := #left_pos_cmd, ref_add := #ref_vel_ramp, fb := #vel_fb, dbw :=, kp := #vel_loop_kp, "T_i[s]" := #"vel_loop_Ti[s]", "T_d[s]" :=, "cycle[s]" := #"cycle[s]", ff_kp := #vel_loop_ff_kp, min := #vel_loop_min, max := #vel_loop_max, cmd => #left_vel_cmd)
   END_RUNG
   // the same network as SCL:
   #pos_loop_Instance_left(run := #run,   // "pos_loop"
                           ref := #ref_pos,
                           fb := #left_pos_fb,
                           dbw := #pos_loop_dbw,
                           Kp := #pos_loop_kp,
                           "T_i[s]" := #"pos_loop_Ti[s]",
                           "cycle[s]" := #"cycle[s]",
                           min := #pos_loop_min,
                           max := #pos_loop_max,
                           cmd => #left_pos_cmd,
                           ENO => #_w1);
   IF #_w1 THEN
       #vel_loop_Instance_left(run := #run,   // "vel_loop"
                               ref := #left_pos_cmd,
                               ref_add := #ref_vel_ramp,
                               fb := #vel_fb,
                               kp := #vel_loop_kp,
                               "T_i[s]" := #"vel_loop_Ti[s]",
                               "cycle[s]" := #"cycle[s]",
                               ff_kp := #vel_loop_ff_kp,
                               min := #vel_loop_min,
                               max := #vel_loop_max,
                               cmd => #left_vel_cmd);
   END_IF;
END_REGION

REGION Network 8
   // feedback velocity = (v1+v2)/2
   RUNG wire#powerrail
      #pos_loop_Instance_right(run := #run, ref := #ref_pos, fb := #right_pos_fb, dbw := #pos_loop_dbw, Kp := #pos_loop_kp, "T_i[s]" := #"pos_loop_Ti[s]", "T_d[s]" :=, "cycle[s]" := #"cycle[s]", min := #pos_loop_min, max := #pos_loop_max, cmd => #right_pos_cmd)
      #vel_loop_Instance_right(run := #run, ref := #right_pos_cmd, ref_add := #ref_vel_ramp, fb := #vel_fb, dbw := #vel_loop_dbw, kp := #vel_loop_kp, "T_i[s]" := #"vel_loop_Ti[s]", "T_d[s]" :=, "cycle[s]" := #"cycle[s]", ff_kp := #vel_loop_ff_kp, min := #vel_loop_min, max := #vel_loop_max, cmd => #right_vel_cmd)
   END_RUNG
   // the same network as SCL:
   #pos_loop_Instance_right(run := #run,   // "pos_loop"
                           ref := #ref_pos,
                           fb := #right_pos_fb,
                           dbw := #pos_loop_dbw,
                           Kp := #pos_loop_kp,
                           "T_i[s]" := #"pos_loop_Ti[s]",
                           "cycle[s]" := #"cycle[s]",
                           min := #pos_loop_min,
                           max := #pos_loop_max,
                           cmd => #right_pos_cmd,
                           ENO => #_w1);
   IF #_w1 THEN
       #vel_loop_Instance_right(run := #run,   // "vel_loop"
                               ref := #right_pos_cmd,
                               ref_add := #ref_vel_ramp,
                               fb := #vel_fb,
                               dbw := #vel_loop_dbw,
                               kp := #vel_loop_kp,
                               "T_i[s]" := #"vel_loop_Ti[s]",
                               "cycle[s]" := #"cycle[s]",
                               ff_kp := #vel_loop_ff_kp,
                               min := #vel_loop_min,
                               max := #vel_loop_max,
                               cmd => #right_vel_cmd);
   END_IF;
END_REGION

REGION Network 9
   RUNG wire#powerrail
      I_Contact( #run )
      Move(in := 0.0, out1 => #ref_vel_ramp)
   END_RUNG
   // the same network as SCL:
   IF NOT #run THEN #ref_vel_ramp := 0.0; END_IF;
END_REGION
END_FUNCTION_BLOCK

FUNCTION_BLOCK "pos_loop"   // FB8, LAD
TITLE = position loop
{ S7_Optimized_Access := 'TRUE' }
VERSION : 0.1
// input:ref_pos, fb_pos
// output: cmd_value
   VAR_INPUT
      run : Bool;
      ref : Real;   // reference
      fb : Real;   // feedback
      dbw : Real;   // deadband width
      Kp : Real;   // proportional factor
      "T_i[s]" : Real;
      "T_d[s]" : Real;
      "cycle[s]" : Real;
      min : Real;
      max : Real;
   END_VAR
   VAR_OUTPUT
      cmd : Real;
   END_VAR
   VAR
      LEAD_LAG_Instance : LEAD_LAG;
      PID_Instance : "PID";
   END_VAR
   VAR_TEMP
      error : Real;
      cmd_b4_out : Real;
      error_deadband : Real;
   END_VAR
   VAR_TEMP   // added for the SCL form of the ladder/FBD networks
      _w1 : Bool;
   END_VAR
BEGIN

REGION Network 1
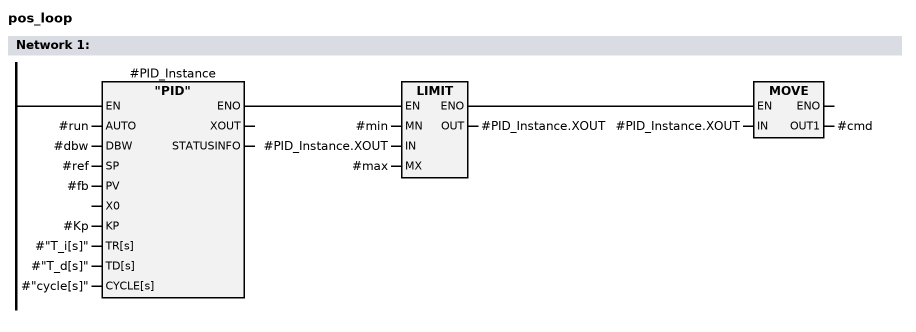
   #PID_Instance(AUTO := #run,   // "PID"
                 DBW := #dbw,
                 SP := #ref,
                 PV := #fb,
                 KP := #Kp,
                 "TR[s]" := #"T_i[s]",
                 "TD[s]" := #"T_d[s]",
                 "CYCLE[s]" := #"cycle[s]",
                 ENO => #_w1);
   IF #_w1 THEN
       #PID_Instance.XOUT := LIMIT(MN := #min, IN := #PID_Instance.XOUT, MX := #max);
       #cmd := #PID_Instance.XOUT;
   END_IF;
END_REGION
END_FUNCTION_BLOCK

FUNCTION_BLOCK "vel_loop"   // FB11, LAD
{ S7_Optimized_Access := 'TRUE' }
VERSION : 0.1
   VAR_INPUT
      run : Bool;
      ref : Real;   // reference
      ref_add : Real;   // additional reference
      fb : Real;   // feedback
      dbw : Real;
      kp : Real;
      "T_i[s]" : Real;
      "T_d[s]" : Real;
      "cycle[s]" : Real;
      ff_kp : Real := 1.0;
      min : Real;
      max : Real;
   END_VAR
   VAR_OUTPUT
      cmd : Real;
   END_VAR
   VAR
      PID_Instance : "PID";
   END_VAR
   VAR_TEMP
      error : Real;
      setpoint : Real;
      pid_out : Real;
      ff_out : Real;
   END_VAR
BEGIN

REGION Network 1
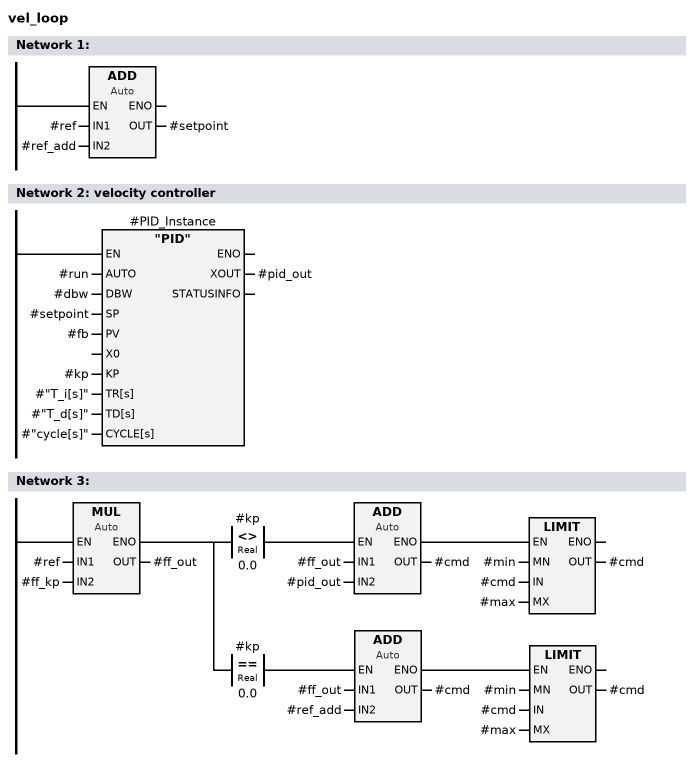
   RUNG wire#powerrail
      Add(in1 := #ref, in2 := #ref_add, out => #setpoint)
   END_RUNG
   // the same network as SCL:
   #setpoint := #ref + #ref_add;
END_REGION

REGION Network 2: velocity controller
   RUNG wire#powerrail
      #PID_Instance(AUTO := #run, DBW := #dbw, SP := #setpoint, PV := #fb, X0 :=, KP := #kp, "TR[s]" := #"T_i[s]", "TD[s]" := #"T_d[s]", "CYCLE[s]" := #"cycle[s]", XOUT => #pid_out, STATUSINFO =>)
   END_RUNG
   // the same network as SCL:
   #PID_Instance(AUTO := #run,   // "PID"
                 DBW := #dbw,
                 SP := #setpoint,
                 PV := #fb,
                 KP := #kp,
                 "TR[s]" := #"T_i[s]",
                 "TD[s]" := #"T_d[s]",
                 "CYCLE[s]" := #"cycle[s]",
                 XOUT => #pid_out);
END_REGION

REGION Network 3
   #ff_out := #ref * #ff_kp;
   IF #kp <> 0.0 THEN
       #cmd := #ff_out + #pid_out;
       #cmd := LIMIT(MN := #min, IN := #cmd, MX := #max);
   END_IF;
   IF #kp = 0.0 THEN
       #cmd := #ff_out + #ref_add;
       #cmd := LIMIT(MN := #min, IN := #cmd, MX := #max);
   END_IF;
END_REGION
END_FUNCTION_BLOCK

FUNCTION "path_planning" : Void   // FC1, LAD
{ S7_Optimized_Access := 'TRUE' }
VERSION : 0.1
// energy sumption optimization
   VAR_INPUT
      IN1 : Real;
      IN2 : Real;
   END_VAR
   VAR_OUTPUT
      OUT : Real;
   END_VAR
BEGIN

REGION Network 1 (SCL)
   #OUT := (#IN1 + #IN2) / 2;
END_REGION
END_FUNCTION

ORGANIZATION_BLOCK "Cyclic_1ms_controller"   // OB31, LAD, CyclicInterrupt
{ S7_Optimized_Access := 'TRUE' }
VERSION : 0.1
   VAR_INPUT
      Initial_Call : Bool;   // Initial call of this OB
      Event_Count : Int;   // Events discarded
   END_VAR
BEGIN

REGION Network 1
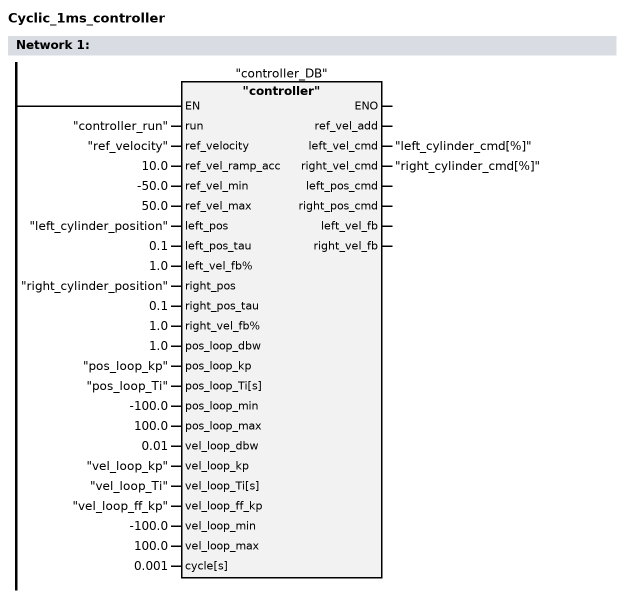
   RUNG wire#powerrail
      "controller_DB"(run := "controller_run", ref_velocity := "ref_velocity", ref_vel_ramp_acc := 10.0, ref_vel_min := -50.0, ref_vel_max := 50.0, left_pos := "left_cylinder_position", left_pos_tau := 0.1, "left_vel_fb%" := 1.0, right_pos := "right_cylinder_position", right_pos_tau := 0.1, "right_vel_fb%" := 1.0, pos_loop_dbw := 1.0, pos_loop_kp := "pos_loop_kp", "pos_loop_Ti[s]" := "pos_loop_Ti", pos_loop_min := -100.0, pos_loop_max := 100.0, vel_loop_dbw := 0.01, vel_loop_kp := "vel_loop_kp", "vel_loop_Ti[s]" := "vel_loop_Ti", vel_loop_ff_kp := "vel_loop_ff_kp", vel_loop_min := -100.0, vel_loop_max := 100.0, "cycle[s]" := 0.001, ref_vel_add =>, left_vel_cmd => "left_cylinder_cmd[%]", right_vel_cmd => "right_cylinder_cmd[%]", left_pos_cmd =>, right_pos_cmd =>, left_vel_fb =>, right_vel_fb =>)
   END_RUNG
   // the same network as SCL:
   "controller_DB"(run := "controller_run",   // "controller"
                   ref_velocity := "ref_velocity",
                   ref_vel_ramp_acc := 10.0,
                   ref_vel_min := -50.0,
                   ref_vel_max := 50.0,
                   left_pos := "left_cylinder_position",
                   left_pos_tau := 0.1,
                   "left_vel_fb%" := 1.0,
                   right_pos := "right_cylinder_position",
                   right_pos_tau := 0.1,
                   "right_vel_fb%" := 1.0,
                   pos_loop_dbw := 1.0,
                   pos_loop_kp := "pos_loop_kp",
                   "pos_loop_Ti[s]" := "pos_loop_Ti",
                   pos_loop_min := -100.0,
                   pos_loop_max := 100.0,
                   vel_loop_dbw := 0.01,
                   vel_loop_kp := "vel_loop_kp",
                   "vel_loop_Ti[s]" := "vel_loop_Ti",
                   vel_loop_ff_kp := "vel_loop_ff_kp",
                   vel_loop_min := -100.0,
                   vel_loop_max := 100.0,
                   "cycle[s]" := 0.001,
                   left_vel_cmd => "left_cylinder_cmd[%]",
                   right_vel_cmd => "right_cylinder_cmd[%]");
END_REGION
END_ORGANIZATION_BLOCK

// folder: ctrl_synch/model

FUNCTION_BLOCK "cylinder"   // FB4, LAD
TITLE = hydraulic cylinder
{ S7_Optimized_Access := 'TRUE' }
VERSION : 0.1
   VAR_INPUT
      run_model : Bool;
      cmd_value : Real;   // command value [%]
      K : Real;   // proportional
      "Tau[s]" : Real;   // delay time [s]
      "T[s]" : Real;   // time constant [s]
      "cycle[s]" : Real;   // scan cycle [s]
      init_pos : Real;   // initial position [mm]
      min_pos : Real;   // min position [mm]
      max_pos : Real := 2000.0;   // max position [mm]
   END_VAR
   VAR_OUTPUT
      velocity : Real;   // [mm/s]
      position : Real;   // [mm]
   END_VAR
   VAR
      DELAY_Instance : "DELAY";
      LAG1_Instance : "LAG1";
      INTEGRAL_Instance : "INTEGRAL";
   END_VAR
   VAR_TEMP
      N_real : Real;
      N_int : Int;   // N time to scan cycle 1ms
      cmd_value_delay : Real;   // command value with delay [%]
      flow_temp : Real;
      velocity_temp : Real;   // [mm/s]
      pos_temp : Real;
   END_VAR
   VAR_TEMP   // added for the SCL form of the ladder/FBD networks
      _w1 : Bool;
   END_VAR
BEGIN

REGION Network 1: Tau
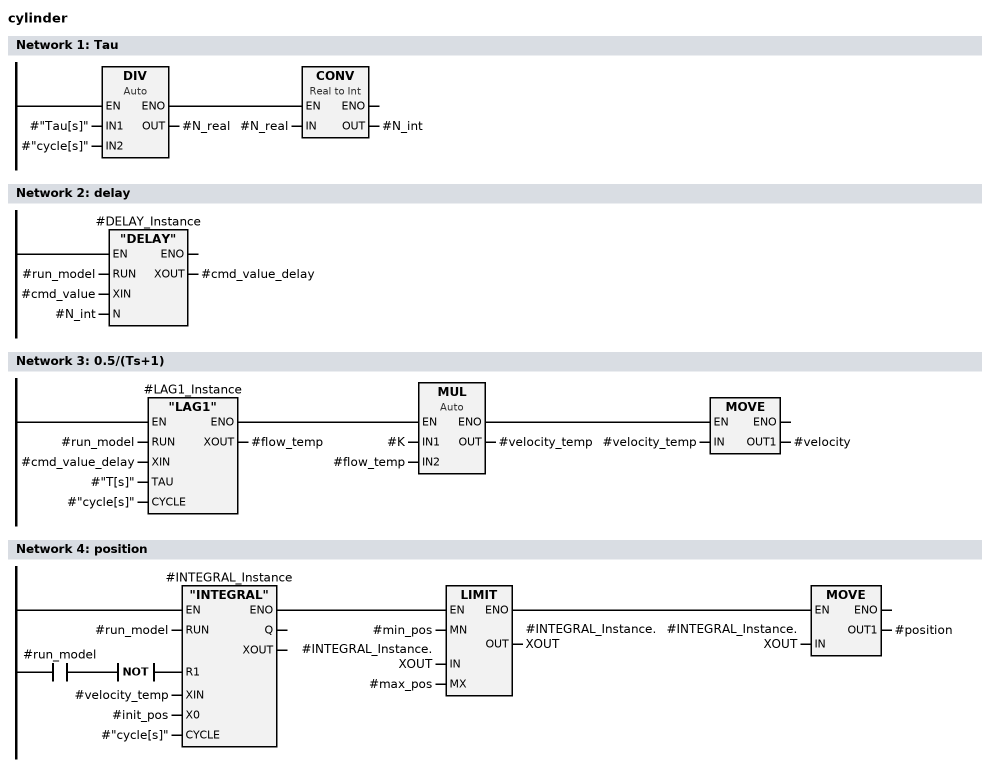
   RUNG wire#powerrail
      Div(in1 := #"Tau[s]", in2 := #"cycle[s]", out => #N_real)
      { S7_Templates := "[SrcType := Real, DestType := Int]" } Convert(in := #N_real, out => #N_int)
   END_RUNG
   // the same network as SCL:
   #N_real := #"Tau[s]" / #"cycle[s]";
   #N_int := REAL_TO_INT(#N_real);
END_REGION

REGION Network 2: delay
   RUNG wire#powerrail
      #DELAY_Instance(RUN := #run_model, XIN := #cmd_value, N := #N_int, XOUT => #cmd_value_delay)
   END_RUNG
   // the same network as SCL:
   #DELAY_Instance(RUN := #run_model, XIN := #cmd_value, N := #N_int, XOUT => #cmd_value_delay);   // "DELAY"
END_REGION

REGION Network 3: 0.5/(Ts+1)
   RUNG wire#powerrail
      #LAG1_Instance(RUN := #run_model, XIN := #cmd_value_delay, TAU := #"T[s]", CYCLE := #"cycle[s]", XOUT => #flow_temp)
      Mul(in1 := #K, in2 := #flow_temp, out => #velocity_temp)
      Move(in := #velocity_temp, out1 => #velocity)
   END_RUNG
   // the same network as SCL:
   #LAG1_Instance(RUN := #run_model,   // "LAG1"
                  XIN := #cmd_value_delay,
                  TAU := #"T[s]",
                  CYCLE := #"cycle[s]",
                  XOUT => #flow_temp,
                  ENO => #_w1);
   IF #_w1 THEN
       #velocity_temp := #K * #flow_temp;
       #velocity := #velocity_temp;
   END_IF;
END_REGION

REGION Network 4: position
   #INTEGRAL_Instance(RUN := #run_model,   // "INTEGRAL"
                      R1 := NOT #run_model,
                      XIN := #velocity_temp,
                      X0 := #init_pos,
                      CYCLE := #"cycle[s]",
                      ENO => #_w1);
   IF #_w1 THEN
       #INTEGRAL_Instance.XOUT := LIMIT(MN := #min_pos, IN := #INTEGRAL_Instance.XOUT, MX := #max_pos);
       #position := #INTEGRAL_Instance.XOUT;
   END_IF;
END_REGION
END_FUNCTION_BLOCK

ORGANIZATION_BLOCK "Cyclic_1ms_model"   // OB30, LAD, CyclicInterrupt
{ S7_Optimized_Access := 'TRUE' }
VERSION : 0.1
   VAR_INPUT
      Initial_Call : Bool;   // Initial call of this OB
      Event_Count : Int;   // Events discarded
   END_VAR
BEGIN

REGION Network 1
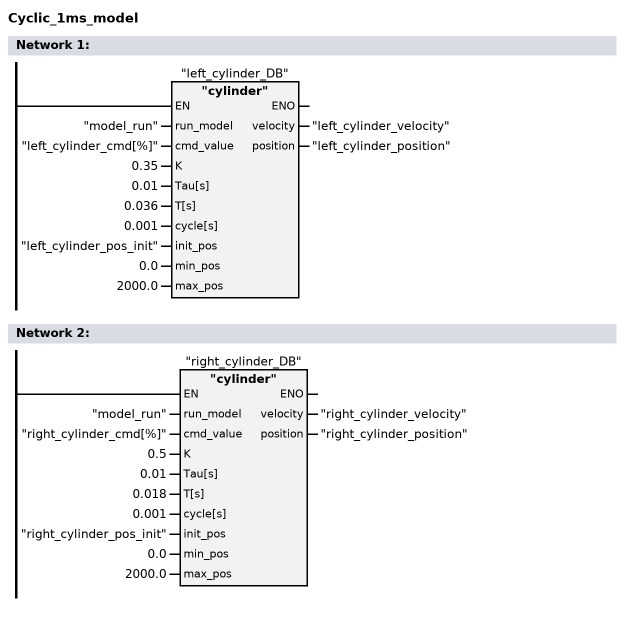
   RUNG wire#powerrail
      "left_cylinder_DB"(run_model := "model_run", cmd_value := "left_cylinder_cmd[%]", K := 0.35, "Tau[s]" := 0.01, "T[s]" := 0.036, "cycle[s]" := 0.001, init_pos := "left_cylinder_pos_init", min_pos := 0.0, max_pos := 2000.0, velocity => "left_cylinder_velocity", position => "left_cylinder_position")
   END_RUNG
   // the same network as SCL:
   "left_cylinder_DB"(run_model := "model_run",   // "cylinder"
                      cmd_value := "left_cylinder_cmd[%]",
                      K := 0.35,
                      "Tau[s]" := 0.01,
                      "T[s]" := 0.036,
                      "cycle[s]" := 0.001,
                      init_pos := "left_cylinder_pos_init",
                      min_pos := 0.0,
                      max_pos := 2000.0,
                      velocity => "left_cylinder_velocity",
                      position => "left_cylinder_position");
END_REGION

REGION Network 2
   RUNG wire#powerrail
      "right_cylinder_DB"(run_model := "model_run", cmd_value := "right_cylinder_cmd[%]", K := 0.5, "Tau[s]" := 0.01, "T[s]" := 0.018, "cycle[s]" := 0.001, init_pos := "right_cylinder_pos_init", min_pos := 0.0, max_pos := 2000.0, velocity => "right_cylinder_velocity", position => "right_cylinder_position")
   END_RUNG
   // the same network as SCL:
   "right_cylinder_DB"(run_model := "model_run",   // "cylinder"
                       cmd_value := "right_cylinder_cmd[%]",
                       K := 0.5,
                       "Tau[s]" := 0.01,
                       "T[s]" := 0.018,
                       "cycle[s]" := 0.001,
                       init_pos := "right_cylinder_pos_init",
                       min_pos := 0.0,
                       max_pos := 2000.0,
                       velocity => "right_cylinder_velocity",
                       position => "right_cylinder_position");
END_REGION
END_ORGANIZATION_BLOCK

// folder: lib

FUNCTION_BLOCK "DELAY"   // FB2, LAD
{ S7_Optimized_Access := 'TRUE' }
VERSION : 0.1
   VAR_INPUT
      RUN : Bool;   // 1 = run, 0 = reset
      XIN : Real;
      N : Int;   // 0 <= N < 128 or specified maximum value
   END_VAR
   VAR_OUTPUT
      XOUT : Real;   // Delayed output
   END_VAR
   VAR
      X : Array[0..127] of Real;   // N-Element queue with FIFO discipline
      I : Int;
      ID : Int;
   END_VAR
BEGIN

REGION Network 1 (SCL)
   IF #RUN THEN
       FOR #ID := 127 TO 1 BY -1 DO
           #X[#ID] := #X[#ID - 1];
       END_FOR;
       #X[0] := #XIN;
       #XOUT := #X[#N];
   ELSE
       #XOUT := #XIN;
       FOR #I := 0 TO #N DO
           #X[#I] := #XIN;
       END_FOR;
   END_IF;
END_REGION
END_FUNCTION_BLOCK

FUNCTION_BLOCK "LAG1"   // FB3, LAD
{ S7_Optimized_Access := 'TRUE' }
VERSION : 0.1
   VAR_INPUT
      RUN : Bool;
      XIN : Real;
      TAU : Real;
      CYCLE : Real;
   END_VAR
   VAR_OUTPUT
      XOUT : Real;
   END_VAR
   VAR
      K : Real;
   END_VAR
BEGIN

REGION Network 1 (SCL)
   IF #RUN THEN
       #XOUT := #XOUT + #K * (#XIN - #XOUT);
   ELSE
       #XOUT := #XIN;
       #K := #CYCLE / (#CYCLE + #TAU);
   END_IF;
END_REGION
END_FUNCTION_BLOCK

FUNCTION_BLOCK "INTEGRAL"   // FB5, LAD
{ S7_Optimized_Access := 'TRUE' }
VERSION : 0.1
   VAR_INPUT
      RUN : Bool;   // 1 = integrate, 0 = hold
      R1 : Bool;   // Overriding reset
      XIN : Real;   // Input variable
      X0 : Real;   // Initial value
      CYCLE : Real;   // Sampling period
   END_VAR
   VAR_OUTPUT
      Q : Bool;   // NOT R1
      XOUT : Real;   // Integrated output
   END_VAR
BEGIN

REGION Network 1 (SCL): NOT R1
   #Q := NOT #R1;
   IF #R1 THEN #XOUT := #X0;
   ELSIF #RUN THEN
       #XOUT := #XOUT + #XIN *#CYCLE;
   END_IF;
END_REGION
END_FUNCTION_BLOCK

FUNCTION_BLOCK "DERIVATIVE"   // FB6, LAD
{ S7_Optimized_Access := 'TRUE' }
VERSION : 0.1
   VAR_INPUT
      RUN : Bool;   // 0 = reset
      XIN : Real;   // Input to be differentiated
      CYCLE : Real;   // Sampling period
   END_VAR
   VAR_OUTPUT
      XOUT : Real;   // Differentiated output
   END_VAR
   VAR
      X1 : Real;
      X2 : Real;
      X3 : Real;
   END_VAR
BEGIN

REGION Network 1 (SCL): Differentiated output
   IF #RUN THEN
       #XOUT := (3.0 * (#XIN - #X3) + #X1 - #X2) / (10.0 * #CYCLE);
       #X3 := #X2;
       #X2 := #X1;
       #X1 := #XIN;
   ELSE
       #XOUT := 0.0;
       #X1 := #XIN;
       #X2 := #XIN;
       #X3 := #XIN;
   END_IF;
END_REGION
END_FUNCTION_BLOCK

FUNCTION_BLOCK "RateLimiter"   // FB9, SCL
{ S7_Optimized_Access := 'TRUE' }
VERSION : 0.1
   VAR_INPUT
      i_R_X : Real;
      i_R_RateLimit : Real;
   END_VAR
   VAR_OUTPUT
      o_R_Y : Real;
   END_VAR
   VAR
      s_R_Y : Real;
      s_R_B4Y : Real;
   END_VAR
   VAR_TEMP
      t_R_Diff : Real;
      t_R_AbsDiff : Real;
      t_R_AbsRateLimit : Real;
      t_R_MinusRateLimit : Real;
   END_VAR
BEGIN

   // Difference = IN - Yn-1
   #t_R_Diff := (#i_R_X - #s_R_B4Y);
   #t_R_AbsDiff := ABS(#t_R_Diff);
   #t_R_AbsRateLimit := ABS(#i_R_RateLimit);
   #t_R_MinusRateLimit := (-1.0) * #i_R_RateLimit;
   // When +|D| ≥ Difference ≥ –|D|: Y = IN
   // When +|D| < Difference: Y = Yn-1 + |D|
   // When –|D| > Difference: Y = Yn-1 - |D|
   IF
       #t_R_AbsDiff <= #t_R_AbsRateLimit
   THEN
       #s_R_Y := #i_R_X;
   ELSIF
       #t_R_AbsRateLimit < #t_R_Diff
   THEN
       #s_R_Y := #s_R_B4Y + #t_R_AbsRateLimit;
   ELSIF
       #t_R_Diff < #t_R_MinusRateLimit
   THEN
       #s_R_Y := #s_R_B4Y - #t_R_AbsRateLimit;
   ELSE
       #s_R_Y := #i_R_X;
   END_IF;
   #s_R_B4Y := #s_R_Y;

   #o_R_Y := #s_R_Y;
END_FUNCTION_BLOCK

FUNCTION_BLOCK "PID"   // FB10, LAD
TITLE = PID Controller
{ S7_Optimized_Access := 'TRUE' }
VERSION : 0.1
// 2021/10/14 Created by GQ
   VAR_INPUT
      AUTO : Bool;   // 0 - manual , 1 - automatic
      DBW : Real;   // Deadband Width
      SP : Real;   // Set point
      PV : Real;   // Process variable
      X0 : Real;   // Manual output adjustment
      KP : Real;   // Proportionality constant
      "TR[s]" : Real;   // Reset time
      "TD[s]" : Real;   // Derivative time constant
      "CYCLE[s]" : Real;   // Sampling period
   END_VAR
   VAR_OUTPUT
      XOUT : Real;
      STATUSINFO : Word;
   END_VAR
   VAR
      ERROR : Real;   // SP-PV
      EDBW : Real;   // ERROR with Deadband
      PIDOUT : Real;
      ITERM : "INTEGRAL";
      DTERM : "DERIVATIVE";
   END_VAR
   VAR CONSTANT
      NO_ERROR : Word := 16#0000;   // No errors
      I_TIME : Word := 16#7000;   // Integral time constant error
      OUT_ARRAY_INDEX : Word := 16#8000;   // Index out of array range
      LIMIT_PARA_FAULT : Word := 16#8200;   // MAX less then MIN in limit
      RATEVALUE_ZERO : Word := 16#8400;   // Rate value zero
   END_VAR
BEGIN

REGION Network 1 (SCL): License
   //=============================================================================
   // (c)Copyright 2021
   //-----------------------------------------------------------------------------
   // Library:       
   // Tested with:   PLCSim Advanced
   // Engineering:   TIA Portal V15 Update 1
   // Restrictions:  
   // Requirements:  PLC (S7-1200 / S7-1500)
   // Functionality: PID Controller for check result of smith predictor
   //-----------------------------------------------------------------------------
   // Change log table:
   // Version  Date        In charge / Changes applied
   // 00.00.01 10.14.2021  002706      created
   //=============================================================================


   IF #"TR[s]" < 0.0 THEN
       #STATUSINFO := #I_TIME;
       RETURN;
   END_IF;

   // IF #MX < #MN THEN
   //     #STATUSINFO := #LIMIT_PARA_FAULT;
   //     RETURN
   //     ;
   // END_IF;

   // IF #RATEVALUE = 0.0 OR #RATEVALUE > (#MX - #MN)THEN
   //     #STATUSINFO := #RATEVALUE_ZERO;
   //     RETURN
   //     ;
   // END_IF;

   #STATUSINFO := #NO_ERROR;
END_REGION

REGION Network 2: ERROR
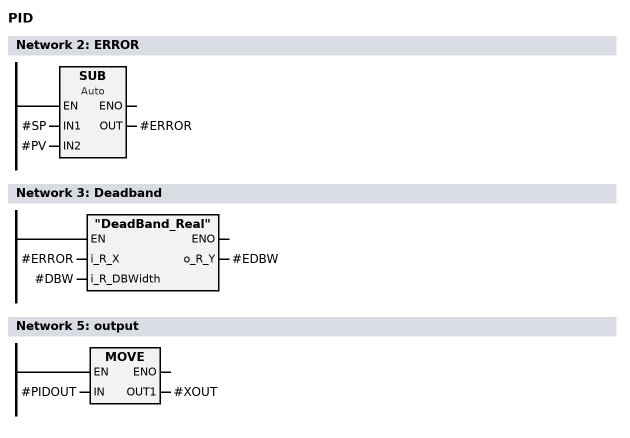
   RUNG wire#powerrail
      Sub(in1 := #SP, in2 := #PV, out => #ERROR)
   END_RUNG
   // the same network as SCL:
   #ERROR := #SP - #PV;
END_REGION

REGION Network 3: Deadband
   RUNG wire#powerrail
      "DeadBand_Real"(i_R_X := #ERROR, i_R_DBWidth := #DBW, o_R_Y => #EDBW)
   END_RUNG
   // the same network as SCL:
   "DeadBand_Real"(i_R_X := #ERROR, i_R_DBWidth := #DBW, o_R_Y => #EDBW);
END_REGION

REGION Network 4 (SCL): PID
   // https://blog.opticontrols.com/archives/383
   // The Cohen-Coon tuning rules were designed for controllers with the noninteractive controller algorithm.
   // Different PID algorithm  equation will cause different result.
   // PID
   (*** Adjust ITERM so that XOUT := X0 when AUTO = 0 ***)
   IF #KP = 0.0 THEN
       #PIDOUT := 0.0;
   ELSE
       #ITERM(RUN := #AUTO,
              R1 := NOT #AUTO,
              XIN := #EDBW,
              X0 := #"TR[s]" * (#X0 - #EDBW),
              CYCLE := #"CYCLE[s]");
       #DTERM(RUN := #AUTO,
              XIN := #EDBW,
              CYCLE := #"CYCLE[s]");
       IF NOT #AUTO THEN
           #PIDOUT := #X0;
       ELSIF #"TR[s]" = 0.0 THEN
           #PIDOUT := #KP * (#EDBW + #DTERM.XOUT * #"TD[s]");
       ELSE
           #PIDOUT := #KP * (#EDBW + #ITERM.XOUT / #"TR[s]" + #DTERM.XOUT * #"TD[s]");
       END_IF;
   END_IF;
END_REGION

REGION Network 5: output
   RUNG wire#powerrail
      Move(in := #PIDOUT, out1 => #XOUT)
   END_RUNG
   // the same network as SCL:
   #XOUT := #PIDOUT;
END_REGION
END_FUNCTION_BLOCK

FUNCTION "LGF_RandomInt" : Int   // FC10013, SCL
{ S7_Optimized_Access := 'TRUE' }
   VAR_INPUT
      minValue : Int;   // minimal Value random can reach
      maxValue : Int;   // maximal Value random can reach
   END_VAR
   VAR_OUTPUT
      error : Bool;
      statusID : UInt;
      status : Word;
   END_VAR
   VAR_TEMP
      tempTime : DTL;
      tempTimeStatus : Int;
      tempRandomValue : Int;
      tempNormReal : Real;
   END_VAR
   VAR CONSTANT
      NO_ERROR : Word := 16#0000;
      NO_CURRENT_JOBS : Word := 16#7000;
      MAX_LESS_MIN : Word := 16#8200;
      ERROR_IN_THIS_BLOCK : UInt := 1;
      ERROR_RD_SYS_T : UInt := 2;
      MIN_INT : DInt := -32768;
      MAX_INT : DInt := 32767;
   END_VAR
BEGIN
   //=============================================================================
   // Siemens AG
   // (c)Copyright 2017
   //-----------------------------------------------------------------------------
   // Library:       LGF (Library General Functions)
   // Tested with:   CPU1212C DC/DC/DC FW:V4.2
   // Engineering:   TIA Portal V13 SP1 Upd 4
   // Restrictions:  -
   // Requirements:  PLC (S7-1200 / S7-1500)
   // Functionality: This function generates random numbers in defined limits
   //                (Datatype Int)
   //-----------------------------------------------------------------------------
   // Change log table:
   // Version  Date        In charge / Changes applied
   // 01.00.00 19.08.2015  Siemens Industry Online Support
   //                      First released version
   // 01.00.01 02.01.2017  Siemens Industry Online Support
   //                      Upgrade: TIA Portal V14 Update 1
   // 01.00.01 10.18.2021  Scale_X 替换成公式 OUT = [VALUE ∗ (MAX – MIN)] + MIN                    
   //-----------------------------------------------------------------------------
   //Status Codes:
   // 16#7000:  No current jobs
   // 16#0000:  Job finished; Note: There is no "Busy"-Status because the block
   //           is finished within a single cycle
   // 16#8200:  maxValue is samller then minValue 
   //=============================================================================

   //Set "No current job" status
   #error := false;
   #statusID := #ERROR_IN_THIS_BLOCK;
   #status := #NO_CURRENT_JOBS;

   //Check if the maximal Value is less than the minimal value
   IF (#minValue > #maxValue) THEN
     #error := true;
     #statusID := #ERROR_IN_THIS_BLOCK;
     #status := #MAX_LESS_MIN;
     #LGF_RandomInt := 0;
     RETURN;
   END_IF;

   //Read system time
   #tempTimeStatus := RD_SYS_T(#tempTime);

   IF (#tempTimeStatus <> 0) THEN
     #error := true;
     #statusID := #ERROR_RD_SYS_T;
     #status := INT_TO_WORD(#tempTimeStatus);
     #LGF_RandomInt := 0;
     RETURN;
   END_IF;

   //Callculate a random-start-value depending on the time
   #tempRandomValue.%B1 := #tempTime.NANOSECOND.%B0;
   #tempRandomValue.%B0 := #tempTime.NANOSECOND.%B1;

   //adapt the calculated random number to the given number span
   #tempNormReal := NORM_X(MIN := #MIN_INT, VALUE := #tempRandomValue, MAX := #MAX_INT);
   // #LGF_RandomInt := SCALE_X(MIN := #minValue, VALUE := #tempNormReal, MAX := #maxValue);
   #LGF_RandomInt := REAL_TO_INT(#tempNormReal * (#maxValue - #minValue) + #minValue);

   #status := #NO_ERROR;
END_FUNCTION

FUNCTION "LGF_RandomReal" : Real   // FC10014, SCL
{ S7_Optimized_Access := 'TRUE' }
   VAR_INPUT
      minValue : Real;   // minimal Value random can reach
      maxValue : Real;   // maximal Value random can reach
   END_VAR
   VAR_OUTPUT
      error : Bool;
      statusID : UInt;
      status : Word;
   END_VAR
   VAR_TEMP
      tempTime : DTL;
      tempTimeStatus : Int;
      tempRandomValue : UDInt;
      tempNormReal : Real;
   END_VAR
   VAR CONSTANT
      NO_ERROR : Word := 16#0000;
      NO_CURRENT_JOBS : Word := 16#7000;
      MAX_LESS_MIN : Word := 16#8200;
      ERROR_IN_THIS_BLOCK : UInt := 1;
      ERROR_RD_SYS_T : UInt := 2;
      MIN_UDINT : UDInt := 0;
      MAX_UDINT : UDInt := 4294967295;
   END_VAR
BEGIN
   //=============================================================================
   // Siemens AG
   // (c)Copyright 2017
   //-----------------------------------------------------------------------------
   // Library:       LGF (Library General Functions)
   // Tested with:   CPU1212C DC/DC/DC FW:V4.2
   // Engineering:   TIA Portal V14 Update 1
   // Restrictions:  -
   // Requirements:  PLC (S7-1200 / S7-1500)
   // Functionality: This function generates random numbers in defined limits
   //                (Datatype Real)
   //-----------------------------------------------------------------------------
   // Change log table:
   // Version  Date        In charge / Changes applied
   // 01.00.00 19.08.2015  Siemens Industry Online Support
   //                      First released version
   // 01.00.01 02.01.2017  Siemens Industry Online Support
   //                      Upgrade: TIA Portal V14 Update 1
   // 01.00.02 02.03.2017  Siemens Industry Online Support
   //                      Bugfix: FC number
   // 01.00.01 10.18.2021  Scale_X 替换成公式 OUT = [VALUE ∗ (MAX – MIN)] + MIN       
   //-----------------------------------------------------------------------------
   //Status Codes:
   // 16#7000:  No current jobs
   // 16#0000:  Job finished   // Note: There is no "Busy"-Status because the
   //           block is finished within a single cycle
   // 16#8200:  maxValue is samller then minValue 
   //=============================================================================

   //Set "No current job" status
   #error := false;
   #statusID := #ERROR_IN_THIS_BLOCK;
   #status := #NO_CURRENT_JOBS;

   //Check if the maximal Value is less than the minimal value
   IF (#minValue > #maxValue) THEN
     #error := true;
     #statusID := #ERROR_IN_THIS_BLOCK;
     #status := #MAX_LESS_MIN;
     #LGF_RandomReal := 0;
     RETURN;
   END_IF;

   //Read system time
   #tempTimeStatus := RD_SYS_T(#tempTime);

   IF (#tempTimeStatus <> 0) THEN
     #error := true;
     #statusID := #ERROR_RD_SYS_T;
     #status := INT_TO_WORD(#tempTimeStatus);
     #LGF_RandomReal := 0;
     RETURN;
   END_IF;

   //Callculate a random-start-value depending on the time
   #tempRandomValue.%B3 := #tempTime.NANOSECOND.%B0;
   #tempRandomValue.%B2 := #tempTime.NANOSECOND.%B1;
   #tempRandomValue.%B1 := #tempTime.NANOSECOND.%B2;
   #tempRandomValue.%B0 := #tempTime.NANOSECOND.%B3;

